//     PlcTask Outputs/GVL_iXlinker.EtherCAT_Master_EPPxxxx.Beckhoff_EPP2xxx.Beckhoff_EPP2xxxEK1122.A_0050_EPP2338_0002_0018.Channel_14.Output <-> Channel 14/Output
//     PlcTask Outputs/GVL_iXlinker.EtherCAT_Master_EPPxxxx.Beckhoff_EPP2xxx.Beckhoff_EPP2xxxEK1122.A_0050_EPP2338_0002_0018.Channel_15.Output <-> Channel 15/Output
//     PlcTask Outputs/GVL_iXlinker.EtherCAT_Master_EPPxxxx.Beckhoff_EPP2xxx.Beckhoff_EPP2xxxEK1122.A_0050_EPP2338_0002_0018.Channel_16.Output <-> Channel 16/Output
//     PlcTask Inputs/GVL_iXlinker.EtherCAT_Master_EPPxxxx.Beckhoff_EPP2xxx.Beckhoff_EPP2xxxEK1122.A_0050_EPP2338_0002_0018.WcState.WcState <-> WcState/WcState
//     PlcTask Inputs/GVL_iXlinker.EtherCAT_Master_EPPxxxx.Beckhoff_EPP2xxx.Beckhoff_EPP2xxxEK1122.A_0050_EPP2338_0002_0018.WcState.InputToggle <-> WcState/InputToggle
//     PlcTask Inputs/GVL_iXlinker.EtherCAT_Master_EPPxxxx.Beckhoff_EPP2xxx.Beckhoff_EPP2xxxEK1122.A_0050_EPP2338_0002_0018.InfoData.State <-> InfoData/State
//   PLC/PLC Instance <-> EtherCAT Master EPPxxxx/Beckhoff EPP2xxx/Beckhoff EPP2xxxEK1122/A_0051(EPP2338-1001-0017)
//     PlcTask Inputs/GVL_iXlinker.EtherCAT_Master_EPPxxxx.Beckhoff_EPP2xxx.Beckhoff_EPP2xxxEK1122.A_0051_EPP2338_1001_0017.Channel_1.Input <-> Channel 1/Input
//     PlcTask Inputs/GVL_iXlinker.EtherCAT_Master_EPPxxxx.Beckhoff_EPP2xxx.Beckhoff_EPP2xxxEK1122.A_0051_EPP2338_1001_0017.Channel_2.Input <-> Channel 2/Input
//     PlcTask Inputs/GVL_iXlinker.EtherCAT_Master_EPPxxxx.Beckhoff_EPP2xxx.Beckhoff_EPP2xxxEK1122.A_0051_EPP2338_1001_0017.Channel_3.Input <-> Channel 3/Input
//     PlcTask Inputs/GVL_iXlinker.EtherCAT_Master_EPPxxxx.Beckhoff_EPP2xxx.Beckhoff_EPP2xxxEK1122.A_0051_EPP2338_1001_0017.Channel_4.Input <-> Channel 4/Input
//     PlcTask Inputs/GVL_iXlinker.EtherCAT_Master_EPPxxxx.Beckhoff_EPP2xxx.Beckhoff_EPP2xxxEK1122.A_0051_EPP2338_1001_0017.Channel_5.Input <-> Channel 5/Input
//     PlcTask Inputs/GVL_iXlinker.EtherCAT_Master_EPPxxxx.Beckhoff_EPP2xxx.Beckhoff_EPP2xxxEK1122.A_0051_EPP2338_1001_0017.Channel_6.Input <-> Channel 6/Input
//     PlcTask Inputs/GVL_iXlinker.EtherCAT_Master_EPPxxxx.Beckhoff_EPP2xxx.Beckhoff_EPP2xxxEK1122.A_0051_EPP2338_1001_0017.Channel_7.Input <-> Channel 7/Input
//     PlcTask Inputs/GVL_iXlinker.EtherCAT_Master_EPPxxxx.Beckhoff_EPP2xxx.Beckhoff_EPP2xxxEK1122.A_0051_EPP2338_1001_0017.Channel_8.Input <-> Channel 8/Input
//     PlcTask Outputs/GVL_iXlinker.EtherCAT_Master_EPPxxxx.Beckhoff_EPP2xxx.Beckhoff_EPP2xxxEK1122.A_0051_EPP2338_1001_0017.Channel_9.Output <-> Channel 9/Output
//     PlcTask Outputs/GVL_iXlinker.EtherCAT_Master_EPPxxxx.Beckhoff_EPP2xxx.Beckhoff_EPP2xxxEK1122.A_0051_EPP2338_1001_0017.Channel_10.Output <-> Channel 10/Output
//     PlcTask Outputs/GVL_iXlinker.EtherCAT_Master_EPPxxxx.Beckhoff_EPP2xxx.Beckhoff_EPP2xxxEK1122.A_0051_EPP2338_1001_0017.Channel_11.Output <-> Channel 11/Output
//     PlcTask Outputs/GVL_iXlinker.EtherCAT_Master_EPPxxxx.Beckhoff_EPP2xxx.Beckhoff_EPP2xxxEK1122.A_0051_EPP2338_1001_0017.Channel_12.Output <-> Channel 12/Output
//     PlcTask Outputs/GVL_iXlinker.EtherCAT_Master_EPPxxxx.Beckhoff_EPP2xxx.Beckhoff_EPP2xxxEK1122.A_0051_EPP2338_1001_0017.Channel_13.Output <-> Channel 13/Output
//     PlcTask Outputs/GVL_iXlinker.EtherCAT_Master_EPPxxxx.Beckhoff_EPP2xxx.Beckhoff_EPP2xxxEK1122.A_0051_EPP2338_1001_0017.Channel_14.Output <-> Channel 14/Output
//     PlcTask Outputs/GVL_iXlinker.EtherCAT_Master_EPPxxxx.Beckhoff_EPP2xxx.Beckhoff_EPP2xxxEK1122.A_0051_EPP2338_1001_0017.Channel_15.Output <-> Channel 15/Output
//     PlcTask Outputs/GVL_iXlinker.EtherCAT_Master_EPPxxxx.Beckhoff_EPP2xxx.Beckhoff_EPP2xxxEK1122.A_0051_EPP2338_1001_0017.Channel_16.Output <-> Channel 16/Output
//     PlcTask Inputs/GVL_iXlinker.EtherCAT_Master_EPPxxxx.Beckhoff_EPP2xxx.Beckhoff_EPP2xxxEK1122.A_0051_EPP2338_1001_0017.WcState.WcState <-> WcState/WcState
//     PlcTask Inputs/GVL_iXlinker.EtherCAT_Master_EPPxxxx.Beckhoff_EPP2xxx.Beckhoff_EPP2xxxEK1122.A_0051_EPP2338_1001_0017.WcState.InputToggle <-> WcState/InputToggle
//     PlcTask Inputs/GVL_iXlinker.EtherCAT_Master_EPPxxxx.Beckhoff_EPP2xxx.Beckhoff_EPP2xxxEK1122.A_0051_EPP2338_1001_0017.InfoData.State <-> InfoData/State
//   PLC/PLC Instance <-> EtherCAT Master EPPxxxx/Beckhoff EPP2xxx/Beckhoff EPP2xxxEK1122/A_0052(EPP2338-1001-0018)
//     PlcTask Inputs/GVL_iXlinker.EtherCAT_Master_EPPxxxx.Beckhoff_EPP2xxx.Beckhoff_EPP2xxxEK1122.A_0052_EPP2338_1001_0018.Channel_1.Input <-> Channel 1/Input
//     PlcTask Inputs/GVL_iXlinker.EtherCAT_Master_EPPxxxx.Beckhoff_EPP2xxx.Beckhoff_EPP2xxxEK1122.A_0052_EPP2338_1001_0018.Channel_2.Input <-> Channel 2/Input
//     PlcTask Inputs/GVL_iXlinker.EtherCAT_Master_EPPxxxx.Beckhoff_EPP2xxx.Beckhoff_EPP2xxxEK1122.A_0052_EPP2338_1001_0018.Channel_3.Input <-> Channel 3/Input
//     PlcTask Inputs/GVL_iXlinker.EtherCAT_Master_EPPxxxx.Beckhoff_EPP2xxx.Beckhoff_EPP2xxxEK1122.A_0052_EPP2338_1001_0018.Channel_4.Input <-> Channel 4/Input
//     PlcTask Inputs/GVL_iXlinker.EtherCAT_Master_EPPxxxx.Beckhoff_EPP2xxx.Beckhoff_EPP2xxxEK1122.A_0052_EPP2338_1001_0018.Channel_5.Input <-> Channel 5/Input
//     PlcTask Inputs/GVL_iXlinker.EtherCAT_Master_EPPxxxx.Beckhoff_EPP2xxx.Beckhoff_EPP2xxxEK1122.A_0052_EPP2338_1001_0018.Channel_6.Input <-> Channel 6/Input
//     PlcTask Inputs/GVL_iXlinker.EtherCAT_Master_EPPxxxx.Beckhoff_EPP2xxx.Beckhoff_EPP2xxxEK1122.A_0052_EPP2338_1001_0018.Channel_7.Input <-> Channel 7/Input
//     PlcTask Inputs/GVL_iXlinker.EtherCAT_Master_EPPxxxx.Beckhoff_EPP2xxx.Beckhoff_EPP2xxxEK1122.A_0052_EPP2338_1001_0018.Channel_8.Input <-> Channel 8/Input
//     PlcTask Outputs/GVL_iXlinker.EtherCAT_Master_EPPxxxx.Beckhoff_EPP2xxx.Beckhoff_EPP2xxxEK1122.A_0052_EPP2338_1001_0018.Channel_9.Output <-> Channel 9/Output
//     PlcTask Outputs/GVL_iXlinker.EtherCAT_Master_EPPxxxx.Beckhoff_EPP2xxx.Beckhoff_EPP2xxxEK1122.A_0052_EPP2338_1001_0018.Channel_10.Output <-> Channel 10/Output
//     PlcTask Outputs/GVL_iXlinker.EtherCAT_Master_EPPxxxx.Beckhoff_EPP2xxx.Beckhoff_EPP2xxxEK1122.A_0052_EPP2338_1001_0018.Channel_11.Output <-> Channel 11/Output
//     PlcTask Outputs/GVL_iXlinker.EtherCAT_Master_EPPxxxx.Beckhoff_EPP2xxx.Beckhoff_EPP2xxxEK1122.A_0052_EPP2338_1001_0018.Channel_12.Output <-> Channel 12/Output
//     PlcTask Outputs/GVL_iXlinker.EtherCAT_Master_EPPxxxx.Beckhoff_EPP2xxx.Beckhoff_EPP2xxxEK1122.A_0052_EPP2338_1001_0018.Channel_13.Output <-> Channel 13/Output
//     PlcTask Outputs/GVL_iXlinker.EtherCAT_Master_EPPxxxx.Beckhoff_EPP2xxx.Beckhoff_EPP2xxxEK1122.A_0052_EPP2338_1001_0018.Channel_14.Output <-> Channel 14/Output
//     PlcTask Outputs/GVL_iXlinker.EtherCAT_Master_EPPxxxx.Beckhoff_EPP2xxx.Beckhoff_EPP2xxxEK1122.A_0052_EPP2338_1001_0018.Channel_15.Output <-> Channel 15/Output
//     PlcTask Outputs/GVL_iXlinker.EtherCAT_Master_EPPxxxx.Beckhoff_EPP2xxx.Beckhoff_EPP2xxxEK1122.A_0052_EPP2338_1001_0018.Channel_16.Output <-> Channel 16/Output
//     PlcTask Inputs/GVL_iXlinker.EtherCAT_Master_EPPxxxx.Beckhoff_EPP2xxx.Beckhoff_EPP2xxxEK1122.A_0052_EPP2338_1001_0018.WcState.WcState <-> WcState/WcState
//     PlcTask Inputs/GVL_iXlinker.EtherCAT_Master_EPPxxxx.Beckhoff_EPP2xxx.Beckhoff_EPP2xxxEK1122.A_0052_EPP2338_1001_0018.WcState.InputToggle <-> WcState/InputToggle
//     PlcTask Inputs/GVL_iXlinker.EtherCAT_Master_EPPxxxx.Beckhoff_EPP2xxx.Beckhoff_EPP2xxxEK1122.A_0052_EPP2338_1001_0018.InfoData.State <-> InfoData/State
//   PLC/PLC Instance <-> EtherCAT Master EPPxxxx/Beckhoff EPP2xxx/Beckhoff EPP2xxxEK1122/A_0053(EPP2338-1001-0019)
//     PlcTask Inputs/GVL_iXlinker.EtherCAT_Master_EPPxxxx.Beckhoff_EPP2xxx.Beckhoff_EPP2xxxEK1122.A_0053_EPP2338_1001_0019.Channel_1.Input <-> Channel 1/Input
//     PlcTask Inputs/GVL_iXlinker.EtherCAT_Master_EPPxxxx.Beckhoff_EPP2xxx.Beckhoff_EPP2xxxEK1122.A_0053_EPP2338_1001_0019.Channel_2.Input <-> Channel 2/Input
//     PlcTask Inputs/GVL_iXlinker.EtherCAT_Master_EPPxxxx.Beckhoff_EPP2xxx.Beckhoff_EPP2xxxEK1122.A_0053_EPP2338_1001_0019.Channel_3.Input <-> Channel 3/Input
//     PlcTask Inputs/GVL_iXlinker.EtherCAT_Master_EPPxxxx.Beckhoff_EPP2xxx.Beckhoff_EPP2xxxEK1122.A_0053_EPP2338_1001_0019.Channel_4.Input <-> Channel 4/Input
//     PlcTask Inputs/GVL_iXlinker.EtherCAT_Master_EPPxxxx.Beckhoff_EPP2xxx.Beckhoff_EPP2xxxEK1122.A_0053_EPP2338_1001_0019.Channel_5.Input <-> Channel 5/Input
//     PlcTask Inputs/GVL_iXlinker.EtherCAT_Master_EPPxxxx.Beckhoff_EPP2xxx.Beckhoff_EPP2xxxEK1122.A_0053_EPP2338_1001_0019.Channel_6.Input <-> Channel 6/Input
//     PlcTask Inputs/GVL_iXlinker.EtherCAT_Master_EPPxxxx.Beckhoff_EPP2xxx.Beckhoff_EPP2xxxEK1122.A_0053_EPP2338_1001_0019.Channel_7.Input <-> Channel 7/Input
//     PlcTask Inputs/GVL_iXlinker.EtherCAT_Master_EPPxxxx.Beckhoff_EPP2xxx.Beckhoff_EPP2xxxEK1122.A_0053_EPP2338_1001_0019.Channel_8.Input <-> Channel 8/Input
//     PlcTask Outputs/GVL_iXlinker.EtherCAT_Master_EPPxxxx.Beckhoff_EPP2xxx.Beckhoff_EPP2xxxEK1122.A_0053_EPP2338_1001_0019.Channel_9.Output <-> Channel 9/Output
//     PlcTask Outputs/GVL_iXlinker.EtherCAT_Master_EPPxxxx.Beckhoff_EPP2xxx.Beckhoff_EPP2xxxEK1122.A_0053_EPP2338_1001_0019.Channel_10.Output <-> Channel 10/Output
//     PlcTask Outputs/GVL_iXlinker.EtherCAT_Master_EPPxxxx.Beckhoff_EPP2xxx.Beckhoff_EPP2xxxEK1122.A_0053_EPP2338_1001_0019.Channel_11.Output <-> Channel 11/Output
//     PlcTask Outputs/GVL_iXlinker.EtherCAT_Master_EPPxxxx.Beckhoff_EPP2xxx.Beckhoff_EPP2xxxEK1122.A_0053_EPP2338_1001_0019.Channel_12.Output <-> Channel 12/Output
//     PlcTask Outputs/GVL_iXlinker.EtherCAT_Master_EPPxxxx.Beckhoff_EPP2xxx.Beckhoff_EPP2xxxEK1122.A_0053_EPP2338_1001_0019.Channel_13.Output <-> Channel 13/Output
//     PlcTask Outputs/GVL_iXlinker.EtherCAT_Master_EPPxxxx.Beckhoff_EPP2xxx.Beckhoff_EPP2xxxEK1122.A_0053_EPP2338_1001_0019.Channel_14.Output <-> Channel 14/Output
//     PlcTask Outputs/GVL_iXlinker.EtherCAT_Master_EPPxxxx.Beckhoff_EPP2xxx.Beckhoff_EPP2xxxEK1122.A_0053_EPP2338_1001_0019.Channel_15.Output <-> Channel 15/Output
//     PlcTask Outputs/GVL_iXlinker.EtherCAT_Master_EPPxxxx.Beckhoff_EPP2xxx.Beckhoff_EPP2xxxEK1122.A_0053_EPP2338_1001_0019.Channel_16.Output <-> Channel 16/Output
//     PlcTask Inputs/GVL_iXlinker.EtherCAT_Master_EPPxxxx.Beckhoff_EPP2xxx.Beckhoff_EPP2xxxEK1122.A_0053_EPP2338_1001_0019.WcState.WcState <-> WcState/WcState
//     PlcTask Inputs/GVL_iXlinker.EtherCAT_Master_EPPxxxx.Beckhoff_EPP2xxx.Beckhoff_EPP2xxxEK1122.A_0053_EPP2338_1001_0019.WcState.InputToggle <-> WcState/InputToggle
//     PlcTask Inputs/GVL_iXlinker.EtherCAT_Master_EPPxxxx.Beckhoff_EPP2xxx.Beckhoff_EPP2xxxEK1122.A_0053_EPP2338_1001_0019.InfoData.State <-> InfoData/State
//   PLC/PLC Instance <-> EtherCAT Master EPPxxxx/Beckhoff EPP2xxx/Beckhoff EPP2xxxEK1122/A_0054(EPP2338-1002-0017)
//     PlcTask Inputs/GVL_iXlinker.EtherCAT_Master_EPPxxxx.Beckhoff_EPP2xxx.Beckhoff_EPP2xxxEK1122.A_0054_EPP2338_1002_0017.Channel_1.Input <-> Channel 1/Input
//     PlcTask Inputs/GVL_iXlinker.EtherCAT_Master_EPPxxxx.Beckhoff_EPP2xxx.Beckhoff_EPP2xxxEK1122.A_0054_EPP2338_1002_0017.Channel_2.Input <-> Channel 2/Input
//     PlcTask Inputs/GVL_iXlinker.EtherCAT_Master_EPPxxxx.Beckhoff_EPP2xxx.Beckhoff_EPP2xxxEK1122.A_0054_EPP2338_1002_0017.Channel_3.Input <-> Channel 3/Input
//     PlcTask Inputs/GVL_iXlinker.EtherCAT_Master_EPPxxxx.Beckhoff_EPP2xxx.Beckhoff_EPP2xxxEK1122.A_0054_EPP2338_1002_0017.Channel_4.Input <-> Channel 4/Input
//     PlcTask Inputs/GVL_iXlinker.EtherCAT_Master_EPPxxxx.Beckhoff_EPP2xxx.Beckhoff_EPP2xxxEK1122.A_0054_EPP2338_1002_0017.Channel_5.Input <-> Channel 5/Input
//     PlcTask Inputs/GVL_iXlinker.EtherCAT_Master_EPPxxxx.Beckhoff_EPP2xxx.Beckhoff_EPP2xxxEK1122.A_0054_EPP2338_1002_0017.Channel_6.Input <-> Channel 6/Input
//     PlcTask Inputs/GVL_iXlinker.EtherCAT_Master_EPPxxxx.Beckhoff_EPP2xxx.Beckhoff_EPP2xxxEK1122.A_0054_EPP2338_1002_0017.Channel_7.Input <-> Channel 7/Input
//     PlcTask Inputs/GVL_iXlinker.EtherCAT_Master_EPPxxxx.Beckhoff_EPP2xxx.Beckhoff_EPP2xxxEK1122.A_0054_EPP2338_1002_0017.Channel_8.Input <-> Channel 8/Input
//     PlcTask Outputs/GVL_iXlinker.EtherCAT_Master_EPPxxxx.Beckhoff_EPP2xxx.Beckhoff_EPP2xxxEK1122.A_0054_EPP2338_1002_0017.Channel_9.Output <-> Channel 9/Output
//     PlcTask Outputs/GVL_iXlinker.EtherCAT_Master_EPPxxxx.Beckhoff_EPP2xxx.Beckhoff_EPP2xxxEK1122.A_0054_EPP2338_1002_0017.Channel_10.Output <-> Channel 10/Output
//     PlcTask Outputs/GVL_iXlinker.EtherCAT_Master_EPPxxxx.Beckhoff_EPP2xxx.Beckhoff_EPP2xxxEK1122.A_0054_EPP2338_1002_0017.Channel_11.Output <-> Channel 11/Output
//     PlcTask Outputs/GVL_iXlinker.EtherCAT_Master_EPPxxxx.Beckhoff_EPP2xxx.Beckhoff_EPP2xxxEK1122.A_0054_EPP2338_1002_0017.Channel_12.Output <-> Channel 12/Output
//     PlcTask Outputs/GVL_iXlinker.EtherCAT_Master_EPPxxxx.Beckhoff_EPP2xxx.Beckhoff_EPP2xxxEK1122.A_0054_EPP2338_1002_0017.Channel_13.Output <-> Channel 13/Output
//     PlcTask Outputs/GVL_iXlinker.EtherCAT_Master_EPPxxxx.Beckhoff_EPP2xxx.Beckhoff_EPP2xxxEK1122.A_0054_EPP2338_1002_0017.Channel_14.Output <-> Channel 14/Output
//     PlcTask Outputs/GVL_iXlinker.EtherCAT_Master_EPPxxxx.Beckhoff_EPP2xxx.Beckhoff_EPP2xxxEK1122.A_0054_EPP2338_1002_0017.Channel_15.Output <-> Channel 15/Output
//     PlcTask Outputs/GVL_iXlinker.EtherCAT_Master_EPPxxxx.Beckhoff_EPP2xxx.Beckhoff_EPP2xxxEK1122.A_0054_EPP2338_1002_0017.Channel_16.Output <-> Channel 16/Output
//     PlcTask Inputs/GVL_iXlinker.EtherCAT_Master_EPPxxxx.Beckhoff_EPP2xxx.Beckhoff_EPP2xxxEK1122.A_0054_EPP2338_1002_0017.WcState.WcState <-> WcState/WcState
//     PlcTask Inputs/GVL_iXlinker.EtherCAT_Master_EPPxxxx.Beckhoff_EPP2xxx.Beckhoff_EPP2xxxEK1122.A_0054_EPP2338_1002_0017.WcState.InputToggle <-> WcState/InputToggle
//     PlcTask Inputs/GVL_iXlinker.EtherCAT_Master_EPPxxxx.Beckhoff_EPP2xxx.Beckhoff_EPP2xxxEK1122.A_0054_EPP2338_1002_0017.InfoData.State <-> InfoData/State
//   PLC/PLC Instance <-> EtherCAT Master EPPxxxx/Beckhoff EPP2xxx/Beckhoff EPP2xxxEK1122/A_0055(EPP2338-1002-0018)
//     PlcTask Inputs/GVL_iXlinker.EtherCAT_Master_EPPxxxx.Beckhoff_EPP2xxx.Beckhoff_EPP2xxxEK1122.A_0055_EPP2338_1002_0018.Channel_1.Input <-> Channel 1/Input
//     PlcTask Inputs/GVL_iXlinker.EtherCAT_Master_EPPxxxx.Beckhoff_EPP2xxx.Beckhoff_EPP2xxxEK1122.A_0055_EPP2338_1002_0018.Channel_2.Input <-> Channel 2/Input
//     PlcTask Inputs/GVL_iXlinker.EtherCAT_Master_EPPxxxx.Beckhoff_EPP2xxx.Beckhoff_EPP2xxxEK1122.A_0055_EPP2338_1002_0018.Channel_3.Input <-> Channel 3/Input
//     PlcTask Inputs/GVL_iXlinker.EtherCAT_Master_EPPxxxx.Beckhoff_EPP2xxx.Beckhoff_EPP2xxxEK1122.A_0055_EPP2338_1002_0018.Channel_4.Input <-> Channel 4/Input
//     PlcTask Inputs/GVL_iXlinker.EtherCAT_Master_EPPxxxx.Beckhoff_EPP2xxx.Beckhoff_EPP2xxxEK1122.A_0055_EPP2338_1002_0018.Channel_5.Input <-> Channel 5/Input
//     PlcTask Inputs/GVL_iXlinker.EtherCAT_Master_EPPxxxx.Beckhoff_EPP2xxx.Beckhoff_EPP2xxxEK1122.A_0055_EPP2338_1002_0018.Channel_6.Input <-> Channel 6/Input
//     PlcTask Inputs/GVL_iXlinker.EtherCAT_Master_EPPxxxx.Beckhoff_EPP2xxx.Beckhoff_EPP2xxxEK1122.A_0055_EPP2338_1002_0018.Channel_7.Input <-> Channel 7/Input
//     PlcTask Inputs/GVL_iXlinker.EtherCAT_Master_EPPxxxx.Beckhoff_EPP2xxx.Beckhoff_EPP2xxxEK1122.A_0055_EPP2338_1002_0018.Channel_8.Input <-> Channel 8/Input
//     PlcTask Outputs/GVL_iXlinker.EtherCAT_Master_EPPxxxx.Beckhoff_EPP2xxx.Beckhoff_EPP2xxxEK1122.A_0055_EPP2338_1002_0018.Channel_9.Output <-> Channel 9/Output
//     PlcTask Outputs/GVL_iXlinker.EtherCAT_Master_EPPxxxx.Beckhoff_EPP2xxx.Beckhoff_EPP2xxxEK1122.A_0055_EPP2338_1002_0018.Channel_10.Output <-> Channel 10/Output
//     PlcTask Outputs/GVL_iXlinker.EtherCAT_Master_EPPxxxx.Beckhoff_EPP2xxx.Beckhoff_EPP2xxxEK1122.A_0055_EPP2338_1002_0018.Channel_11.Output <-> Channel 11/Output
//     PlcTask Outputs/GVL_iXlinker.EtherCAT_Master_EPPxxxx.Beckhoff_EPP2xxx.Beckhoff_EPP2xxxEK1122.A_0055_EPP2338_1002_0018.Channel_12.Output <-> Channel 12/Output
//     PlcTask Outputs/GVL_iXlinker.EtherCAT_Master_EPPxxxx.Beckhoff_EPP2xxx.Beckhoff_EPP2xxxEK1122.A_0055_EPP2338_1002_0018.Channel_13.Output <-> Channel 13/Output
//     PlcTask Outputs/GVL_iXlinker.EtherCAT_Master_EPPxxxx.Beckhoff_EPP2xxx.Beckhoff_EPP2xxxEK1122.A_0055_EPP2338_1002_0018.Channel_14.Output <-> Channel 14/Output
//     PlcTask Outputs/GVL_iXlinker.EtherCAT_Master_EPPxxxx.Beckhoff_EPP2xxx.Beckhoff_EPP2xxxEK1122.A_0055_EPP2338_1002_0018.Channel_15.Output <-> Channel 15/Output
//     PlcTask Outputs/GVL_iXlinker.EtherCAT_Master_EPPxxxx.Beckhoff_EPP2xxx.Beckhoff_EPP2xxxEK1122.A_0055_EPP2338_1002_0018.Channel_16.Output <-> Channel 16/Output
//     PlcTask Inputs/GVL_iXlinker.EtherCAT_Master_EPPxxxx.Beckhoff_EPP2xxx.Beckhoff_EPP2xxxEK1122.A_0055_EPP2338_1002_0018.WcState.WcState <-> WcState/WcState
//     PlcTask Inputs/GVL_iXlinker.EtherCAT_Master_EPPxxxx.Beckhoff_EPP2xxx.Beckhoff_EPP2xxxEK1122.A_0055_EPP2338_1002_0018.WcState.InputToggle <-> WcState/InputToggle
//     PlcTask Inputs/GVL_iXlinker.EtherCAT_Master_EPPxxxx.Beckhoff_EPP2xxx.Beckhoff_EPP2xxxEK1122.A_0055_EPP2338_1002_0018.InfoData.State <-> InfoData/State
//   PLC/PLC Instance <-> EtherCAT Master EPPxxxx/Beckhoff EPP2xxx/Beckhoff EPP2xxxEK1122/A_0056(EPP2338-1002-0019)
//     PlcTask Inputs/GVL_iXlinker.EtherCAT_Master_EPPxxxx.Beckhoff_EPP2xxx.Beckhoff_EPP2xxxEK1122.A_0056_EPP2338_1002_0019.Channel_1.Input <-> Channel 1/Input
//     PlcTask Inputs/GVL_iXlinker.EtherCAT_Master_EPPxxxx.Beckhoff_EPP2xxx.Beckhoff_EPP2xxxEK1122.A_0056_EPP2338_1002_0019.Channel_2.Input <-> Channel 2/Input
//     PlcTask Inputs/GVL_iXlinker.EtherCAT_Master_EPPxxxx.Beckhoff_EPP2xxx.Beckhoff_EPP2xxxEK1122.A_0056_EPP2338_1002_0019.Channel_3.Input <-> Channel 3/Input
//     PlcTask Inputs/GVL_iXlinker.EtherCAT_Master_EPPxxxx.Beckhoff_EPP2xxx.Beckhoff_EPP2xxxEK1122.A_0056_EPP2338_1002_0019.Channel_4.Input <-> Channel 4/Input
//     PlcTask Inputs/GVL_iXlinker.EtherCAT_Master_EPPxxxx.Beckhoff_EPP2xxx.Beckhoff_EPP2xxxEK1122.A_0056_EPP2338_1002_0019.Channel_5.Input <-> Channel 5/Input
//     PlcTask Inputs/GVL_iXlinker.EtherCAT_Master_EPPxxxx.Beckhoff_EPP2xxx.Beckhoff_EPP2xxxEK1122.A_0056_EPP2338_1002_0019.Channel_6.Input <-> Channel 6/Input
//     PlcTask Inputs/GVL_iXlinker.EtherCAT_Master_EPPxxxx.Beckhoff_EPP2xxx.Beckhoff_EPP2xxxEK1122.A_0056_EPP2338_1002_0019.Channel_7.Input <-> Channel 7/Input
//     PlcTask Inputs/GVL_iXlinker.EtherCAT_Master_EPPxxxx.Beckhoff_EPP2xxx.Beckhoff_EPP2xxxEK1122.A_0056_EPP2338_1002_0019.Channel_8.Input <-> Channel 8/Input
//     PlcTask Outputs/GVL_iXlinker.EtherCAT_Master_EPPxxxx.Beckhoff_EPP2xxx.Beckhoff_EPP2xxxEK1122.A_0056_EPP2338_1002_0019.Channel_9.Output <-> Channel 9/Output
//     PlcTask Outputs/GVL_iXlinker.EtherCAT_Master_EPPxxxx.Beckhoff_EPP2xxx.Beckhoff_EPP2xxxEK1122.A_0056_EPP2338_1002_0019.Channel_10.Output <-> Channel 10/Output
//     PlcTask Outputs/GVL_iXlinker.EtherCAT_Master_EPPxxxx.Beckhoff_EPP2xxx.Beckhoff_EPP2xxxEK1122.A_0056_EPP2338_1002_0019.Channel_11.Output <-> Channel 11/Output
//     PlcTask Outputs/GVL_iXlinker.EtherCAT_Master_EPPxxxx.Beckhoff_EPP2xxx.Beckhoff_EPP2xxxEK1122.A_0056_EPP2338_1002_0019.Channel_12.Output <-> Channel 12/Output
//     PlcTask Outputs/GVL_iXlinker.EtherCAT_Master_EPPxxxx.Beckhoff_EPP2xxx.Beckhoff_EPP2xxxEK1122.A_0056_EPP2338_1002_0019.Channel_13.Output <-> Channel 13/Output
//     PlcTask Outputs/GVL_iXlinker.EtherCAT_Master_EPPxxxx.Beckhoff_EPP2xxx.Beckhoff_EPP2xxxEK1122.A_0056_EPP2338_1002_0019.Channel_14.Output <-> Channel 14/Output
//     PlcTask Outputs/GVL_iXlinker.EtherCAT_Master_EPPxxxx.Beckhoff_EPP2xxx.Beckhoff_EPP2xxxEK1122.A_0056_EPP2338_1002_0019.Channel_15.Output <-> Channel 15/Output
//     PlcTask Outputs/GVL_iXlinker.EtherCAT_Master_EPPxxxx.Beckhoff_EPP2xxx.Beckhoff_EPP2xxxEK1122.A_0056_EPP2338_1002_0019.Channel_16.Output <-> Channel 16/Output
//     PlcTask Inputs/GVL_iXlinker.EtherCAT_Master_EPPxxxx.Beckhoff_EPP2xxx.Beckhoff_EPP2xxxEK1122.A_0056_EPP2338_1002_0019.WcState.WcState <-> WcState/WcState
//     PlcTask Inputs/GVL_iXlinker.EtherCAT_Master_EPPxxxx.Beckhoff_EPP2xxx.Beckhoff_EPP2xxxEK1122.A_0056_EPP2338_1002_0019.WcState.InputToggle <-> WcState/InputToggle
//     PlcTask Inputs/GVL_iXlinker.EtherCAT_Master_EPPxxxx.Beckhoff_EPP2xxx.Beckhoff_EPP2xxxEK1122.A_0056_EPP2338_1002_0019.InfoData.State <-> InfoData/State
//   PLC/PLC Instance <-> EtherCAT Master EPPxxxx/Beckhoff EPP2xxx/Beckhoff EPP2xxxEK1122/A_0057(EPP2339-0003-0016)
//     PlcTask Inputs/GVL_iXlinker.EtherCAT_Master_EPPxxxx.Beckhoff_EPP2xxx.Beckhoff_EPP2xxxEK1122.A_0057_EPP2339_0003_0016.DI_Inputs_Channel_1.Input[0] <-> DI Inputs Channel 1/Input 1
//     PlcTask Inputs/GVL_iXlinker.EtherCAT_Master_EPPxxxx.Beckhoff_EPP2xxx.Beckhoff_EPP2xxxEK1122.A_0057_EPP2339_0003_0016.DI_Inputs_Channel_1.Input[1] <-> DI Inputs Channel 1/Input 2
//     PlcTask Inputs/GVL_iXlinker.EtherCAT_Master_EPPxxxx.Beckhoff_EPP2xxx.Beckhoff_EPP2xxxEK1122.A_0057_EPP2339_0003_0016.DI_Inputs_Channel_1.Input[2] <-> DI Inputs Channel 1/Input 3
//     PlcTask Inputs/GVL_iXlinker.EtherCAT_Master_EPPxxxx.Beckhoff_EPP2xxx.Beckhoff_EPP2xxxEK1122.A_0057_EPP2339_0003_0016.DI_Inputs_Channel_1.Input[3] <-> DI Inputs Channel 1/Input 4
//     PlcTask Inputs/GVL_iXlinker.EtherCAT_Master_EPPxxxx.Beckhoff_EPP2xxx.Beckhoff_EPP2xxxEK1122.A_0057_EPP2339_0003_0016.DI_Inputs_Channel_1.Input[4] <-> DI Inputs Channel 1/Input 5
//     PlcTask Inputs/GVL_iXlinker.EtherCAT_Master_EPPxxxx.Beckhoff_EPP2xxx.Beckhoff_EPP2xxxEK1122.A_0057_EPP2339_0003_0016.DI_Inputs_Channel_1.Input[5] <-> DI Inputs Channel 1/Input 6
//     PlcTask Inputs/GVL_iXlinker.EtherCAT_Master_EPPxxxx.Beckhoff_EPP2xxx.Beckhoff_EPP2xxxEK1122.A_0057_EPP2339_0003_0016.DI_Inputs_Channel_1.Input[6] <-> DI Inputs Channel 1/Input 7
//     PlcTask Inputs/GVL_iXlinker.EtherCAT_Master_EPPxxxx.Beckhoff_EPP2xxx.Beckhoff_EPP2xxxEK1122.A_0057_EPP2339_0003_0016.DI_Inputs_Channel_1.Input[7] <-> DI Inputs Channel 1/Input 8
//     PlcTask Inputs/GVL_iXlinker.EtherCAT_Master_EPPxxxx.Beckhoff_EPP2xxx.Beckhoff_EPP2xxxEK1122.A_0057_EPP2339_0003_0016.DI_Inputs_Channel_2.Input[0] <-> DI Inputs Channel 2/Input 1
//     PlcTask Inputs/GVL_iXlinker.EtherCAT_Master_EPPxxxx.Beckhoff_EPP2xxx.Beckhoff_EPP2xxxEK1122.A_0057_EPP2339_0003_0016.DI_Inputs_Channel_2.Input[1] <-> DI Inputs Channel 2/Input 2
//     PlcTask Inputs/GVL_iXlinker.EtherCAT_Master_EPPxxxx.Beckhoff_EPP2xxx.Beckhoff_EPP2xxxEK1122.A_0057_EPP2339_0003_0016.DI_Inputs_Channel_2.Input[2] <-> DI Inputs Channel 2/Input 3
//     PlcTask Inputs/GVL_iXlinker.EtherCAT_Master_EPPxxxx.Beckhoff_EPP2xxx.Beckhoff_EPP2xxxEK1122.A_0057_EPP2339_0003_0016.DI_Inputs_Channel_2.Input[3] <-> DI Inputs Channel 2/Input 4
//     PlcTask Inputs/GVL_iXlinker.EtherCAT_Master_EPPxxxx.Beckhoff_EPP2xxx.Beckhoff_EPP2xxxEK1122.A_0057_EPP2339_0003_0016.DI_Inputs_Channel_2.Input[4] <-> DI Inputs Channel 2/Input 5
//     PlcTask Inputs/GVL_iXlinker.EtherCAT_Master_EPPxxxx.Beckhoff_EPP2xxx.Beckhoff_EPP2xxxEK1122.A_0057_EPP2339_0003_0016.DI_Inputs_Channel_2.Input[5] <-> DI Inputs Channel 2/Input 6
//     PlcTask Inputs/GVL_iXlinker.EtherCAT_Master_EPPxxxx.Beckhoff_EPP2xxx.Beckhoff_EPP2xxxEK1122.A_0057_EPP2339_0003_0016.DI_Inputs_Channel_2.Input[6] <-> DI Inputs Channel 2/Input 7
//     PlcTask Inputs/GVL_iXlinker.EtherCAT_Master_EPPxxxx.Beckhoff_EPP2xxx.Beckhoff_EPP2xxxEK1122.A_0057_EPP2339_0003_0016.DI_Inputs_Channel_2.Input[7] <-> DI Inputs Channel 2/Input 8
//     PlcTask Inputs/GVL_iXlinker.EtherCAT_Master_EPPxxxx.Beckhoff_EPP2xxx.Beckhoff_EPP2xxxEK1122.A_0057_EPP2339_0003_0016.DI_Inputs_Channel_1.Sync_error <-> DI Inputs Channel 1/Sync error
//     PlcTask Inputs/GVL_iXlinker.EtherCAT_Master_EPPxxxx.Beckhoff_EPP2xxx.Beckhoff_EPP2xxxEK1122.A_0057_EPP2339_0003_0016.DI_Inputs_Channel_2.Sync_error <-> DI Inputs Channel 2/Sync error
//     PlcTask Inputs/GVL_iXlinker.EtherCAT_Master_EPPxxxx.Beckhoff_EPP2xxx.Beckhoff_EPP2xxxEK1122.A_0057_EPP2339_0003_0016.DI_Inputs_Channel_1.TxPDO_State <-> DI Inputs Channel 1/TxPDO State
//     PlcTask Inputs/GVL_iXlinker.EtherCAT_Master_EPPxxxx.Beckhoff_EPP2xxx.Beckhoff_EPP2xxxEK1122.A_0057_EPP2339_0003_0016.DI_Inputs_Channel_2.TxPDO_State <-> DI Inputs Channel 2/TxPDO State
//     PlcTask Inputs/GVL_iXlinker.EtherCAT_Master_EPPxxxx.Beckhoff_EPP2xxx.Beckhoff_EPP2xxxEK1122.A_0057_EPP2339_0003_0016.DI_Inputs_Channel_1.TxPDO_Toggle <-> DI Inputs Channel 1/TxPDO Toggle
//     PlcTask Inputs/GVL_iXlinker.EtherCAT_Master_EPPxxxx.Beckhoff_EPP2xxx.Beckhoff_EPP2xxxEK1122.A_0057_EPP2339_0003_0016.DI_Inputs_Channel_2.TxPDO_Toggle <-> DI Inputs Channel 2/TxPDO Toggle
//     PlcTask Outputs/GVL_iXlinker.EtherCAT_Master_EPPxxxx.Beckhoff_EPP2xxx.Beckhoff_EPP2xxxEK1122.A_0057_EPP2339_0003_0016.DO_Outputs_Channel_1.Output[0] <-> DO Outputs Channel 1/Output 1
//     PlcTask Outputs/GVL_iXlinker.EtherCAT_Master_EPPxxxx.Beckhoff_EPP2xxx.Beckhoff_EPP2xxxEK1122.A_0057_EPP2339_0003_0016.DO_Outputs_Channel_1.Output[1] <-> DO Outputs Channel 1/Output 2
//     PlcTask Outputs/GVL_iXlinker.EtherCAT_Master_EPPxxxx.Beckhoff_EPP2xxx.Beckhoff_EPP2xxxEK1122.A_0057_EPP2339_0003_0016.DO_Outputs_Channel_1.Output[2] <-> DO Outputs Channel 1/Output 3
//     PlcTask Outputs/GVL_iXlinker.EtherCAT_Master_EPPxxxx.Beckhoff_EPP2xxx.Beckhoff_EPP2xxxEK1122.A_0057_EPP2339_0003_0016.DO_Outputs_Channel_1.Output[3] <-> DO Outputs Channel 1/Output 4
//     PlcTask Outputs/GVL_iXlinker.EtherCAT_Master_EPPxxxx.Beckhoff_EPP2xxx.Beckhoff_EPP2xxxEK1122.A_0057_EPP2339_0003_0016.DO_Outputs_Channel_1.Output[4] <-> DO Outputs Channel 1/Output 5
//     PlcTask Outputs/GVL_iXlinker.EtherCAT_Master_EPPxxxx.Beckhoff_EPP2xxx.Beckhoff_EPP2xxxEK1122.A_0057_EPP2339_0003_0016.DO_Outputs_Channel_1.Output[5] <-> DO Outputs Channel 1/Output 6
//     PlcTask Outputs/GVL_iXlinker.EtherCAT_Master_EPPxxxx.Beckhoff_EPP2xxx.Beckhoff_EPP2xxxEK1122.A_0057_EPP2339_0003_0016.DO_Outputs_Channel_1.Output[6] <-> DO Outputs Channel 1/Output 7
//     PlcTask Outputs/GVL_iXlinker.EtherCAT_Master_EPPxxxx.Beckhoff_EPP2xxx.Beckhoff_EPP2xxxEK1122.A_0057_EPP2339_0003_0016.DO_Outputs_Channel_1.Output[7] <-> DO Outputs Channel 1/Output 8
//     PlcTask Outputs/GVL_iXlinker.EtherCAT_Master_EPPxxxx.Beckhoff_EPP2xxx.Beckhoff_EPP2xxxEK1122.A_0057_EPP2339_0003_0016.DO_Outputs_Channel_2.Output[0] <-> DO Outputs Channel 2/Output 1
//     PlcTask Outputs/GVL_iXlinker.EtherCAT_Master_EPPxxxx.Beckhoff_EPP2xxx.Beckhoff_EPP2xxxEK1122.A_0057_EPP2339_0003_0016.DO_Outputs_Channel_2.Output[1] <-> DO Outputs Channel 2/Output 2
//     PlcTask Outputs/GVL_iXlinker.EtherCAT_Master_EPPxxxx.Beckhoff_EPP2xxx.Beckhoff_EPP2xxxEK1122.A_0057_EPP2339_0003_0016.DO_Outputs_Channel_2.Output[2] <-> DO Outputs Channel 2/Output 3
//     PlcTask Outputs/GVL_iXlinker.EtherCAT_Master_EPPxxxx.Beckhoff_EPP2xxx.Beckhoff_EPP2xxxEK1122.A_0057_EPP2339_0003_0016.DO_Outputs_Channel_2.Output[3] <-> DO Outputs Channel 2/Output 4
//     PlcTask Outputs/GVL_iXlinker.EtherCAT_Master_EPPxxxx.Beckhoff_EPP2xxx.Beckhoff_EPP2xxxEK1122.A_0057_EPP2339_0003_0016.DO_Outputs_Channel_2.Output[4] <-> DO Outputs Channel 2/Output 5
//     PlcTask Outputs/GVL_iXlinker.EtherCAT_Master_EPPxxxx.Beckhoff_EPP2xxx.Beckhoff_EPP2xxxEK1122.A_0057_EPP2339_0003_0016.DO_Outputs_Channel_2.Output[5] <-> DO Outputs Channel 2/Output 6
//     PlcTask Outputs/GVL_iXlinker.EtherCAT_Master_EPPxxxx.Beckhoff_EPP2xxx.Beckhoff_EPP2xxxEK1122.A_0057_EPP2339_0003_0016.DO_Outputs_Channel_2.Output[6] <-> DO Outputs Channel 2/Output 7
//     PlcTask Outputs/GVL_iXlinker.EtherCAT_Master_EPPxxxx.Beckhoff_EPP2xxx.Beckhoff_EPP2xxxEK1122.A_0057_EPP2339_0003_0016.DO_Outputs_Channel_2.Output[7] <-> DO Outputs Channel 2/Output 8
//     PlcTask Inputs/GVL_iXlinker.EtherCAT_Master_EPPxxxx.Beckhoff_EPP2xxx.Beckhoff_EPP2xxxEK1122.A_0057_EPP2339_0003_0016.WcState.WcState <-> WcState/WcState
//     PlcTask Inputs/GVL_iXlinker.EtherCAT_Master_EPPxxxx.Beckhoff_EPP2xxx.Beckhoff_EPP2xxxEK1122.A_0057_EPP2339_0003_0016.WcState.InputToggle <-> WcState/InputToggle
//     PlcTask Inputs/GVL_iXlinker.EtherCAT_Master_EPPxxxx.Beckhoff_EPP2xxx.Beckhoff_EPP2xxxEK1122.A_0057_EPP2339_0003_0016.InfoData.AdsAddr <-> InfoData/AdsAddr
//     PlcTask Inputs/GVL_iXlinker.EtherCAT_Master_EPPxxxx.Beckhoff_EPP2xxx.Beckhoff_EPP2xxxEK1122.A_0057_EPP2339_0003_0016.InfoData.State <-> InfoData/State
//   PLC/PLC Instance <-> EtherCAT Master EPPxxxx/Beckhoff EPP2xxx/Beckhoff EPP2xxxEK1122/A_0058(EPP2339-0021-0016)
//     PlcTask Inputs/GVL_iXlinker.EtherCAT_Master_EPPxxxx.Beckhoff_EPP2xxx.Beckhoff_EPP2xxxEK1122.A_0058_EPP2339_0021_0016.Channel_1.Input <-> Channel 1/Input
//     PlcTask Inputs/GVL_iXlinker.EtherCAT_Master_EPPxxxx.Beckhoff_EPP2xxx.Beckhoff_EPP2xxxEK1122.A_0058_EPP2339_0021_0016.Channel_2.Input <-> Channel 2/Input
//     PlcTask Inputs/GVL_iXlinker.EtherCAT_Master_EPPxxxx.Beckhoff_EPP2xxx.Beckhoff_EPP2xxxEK1122.A_0058_EPP2339_0021_0016.Channel_3.Input <-> Channel 3/Input
//     PlcTask Inputs/GVL_iXlinker.EtherCAT_Master_EPPxxxx.Beckhoff_EPP2xxx.Beckhoff_EPP2xxxEK1122.A_0058_EPP2339_0021_0016.Channel_4.Input <-> Channel 4/Input
//     PlcTask Inputs/GVL_iXlinker.EtherCAT_Master_EPPxxxx.Beckhoff_EPP2xxx.Beckhoff_EPP2xxxEK1122.A_0058_EPP2339_0021_0016.Channel_5.Input <-> Channel 5/Input
//     PlcTask Inputs/GVL_iXlinker.EtherCAT_Master_EPPxxxx.Beckhoff_EPP2xxx.Beckhoff_EPP2xxxEK1122.A_0058_EPP2339_0021_0016.Channel_6.Input <-> Channel 6/Input
//     PlcTask Inputs/GVL_iXlinker.EtherCAT_Master_EPPxxxx.Beckhoff_EPP2xxx.Beckhoff_EPP2xxxEK1122.A_0058_EPP2339_0021_0016.Channel_7.Input <-> Channel 7/Input
//     PlcTask Inputs/GVL_iXlinker.EtherCAT_Master_EPPxxxx.Beckhoff_EPP2xxx.Beckhoff_EPP2xxxEK1122.A_0058_EPP2339_0021_0016.Channel_8.Input <-> Channel 8/Input
//     PlcTask Inputs/GVL_iXlinker.EtherCAT_Master_EPPxxxx.Beckhoff_EPP2xxx.Beckhoff_EPP2xxxEK1122.A_0058_EPP2339_0021_0016.Channel_9.Input <-> Channel 9/Input
//     PlcTask Inputs/GVL_iXlinker.EtherCAT_Master_EPPxxxx.Beckhoff_EPP2xxx.Beckhoff_EPP2xxxEK1122.A_0058_EPP2339_0021_0016.Channel_10.Input <-> Channel 10/Input
//     PlcTask Inputs/GVL_iXlinker.EtherCAT_Master_EPPxxxx.Beckhoff_EPP2xxx.Beckhoff_EPP2xxxEK1122.A_0058_EPP2339_0021_0016.Channel_11.Input <-> Channel 11/Input
//     PlcTask Inputs/GVL_iXlinker.EtherCAT_Master_EPPxxxx.Beckhoff_EPP2xxx.Beckhoff_EPP2xxxEK1122.A_0058_EPP2339_0021_0016.Channel_12.Input <-> Channel 12/Input
//     PlcTask Inputs/GVL_iXlinker.EtherCAT_Master_EPPxxxx.Beckhoff_EPP2xxx.Beckhoff_EPP2xxxEK1122.A_0058_EPP2339_0021_0016.Channel_13.Input <-> Channel 13/Input
//     PlcTask Inputs/GVL_iXlinker.EtherCAT_Master_EPPxxxx.Beckhoff_EPP2xxx.Beckhoff_EPP2xxxEK1122.A_0058_EPP2339_0021_0016.Channel_14.Input <-> Channel 14/Input
//     PlcTask Inputs/GVL_iXlinker.EtherCAT_Master_EPPxxxx.Beckhoff_EPP2xxx.Beckhoff_EPP2xxxEK1122.A_0058_EPP2339_0021_0016.Channel_15.Input <-> Channel 15/Input
//     PlcTask Inputs/GVL_iXlinker.EtherCAT_Master_EPPxxxx.Beckhoff_EPP2xxx.Beckhoff_EPP2xxxEK1122.A_0058_EPP2339_0021_0016.Channel_16.Input <-> Channel 16/Input
//     PlcTask Outputs/GVL_iXlinker.EtherCAT_Master_EPPxxxx.Beckhoff_EPP2xxx.Beckhoff_EPP2xxxEK1122.A_0058_EPP2339_0021_0016.Channel_9_1.Output <-> Channel 9_1/Output
//     PlcTask Outputs/GVL_iXlinker.EtherCAT_Master_EPPxxxx.Beckhoff_EPP2xxx.Beckhoff_EPP2xxxEK1122.A_0058_EPP2339_0021_0016.Channel_10_1.Output <-> Channel 10_1/Output
//     PlcTask Outputs/GVL_iXlinker.EtherCAT_Master_EPPxxxx.Beckhoff_EPP2xxx.Beckhoff_EPP2xxxEK1122.A_0058_EPP2339_0021_0016.Channel_11_1.Output <-> Channel 11_1/Output
//     PlcTask Outputs/GVL_iXlinker.EtherCAT_Master_EPPxxxx.Beckhoff_EPP2xxx.Beckhoff_EPP2xxxEK1122.A_0058_EPP2339_0021_0016.Channel_12_1.Output <-> Channel 12_1/Output
//     PlcTask Outputs/GVL_iXlinker.EtherCAT_Master_EPPxxxx.Beckhoff_EPP2xxx.Beckhoff_EPP2xxxEK1122.A_0058_EPP2339_0021_0016.Channel_13_1.Output <-> Channel 13_1/Output
//     PlcTask Outputs/GVL_iXlinker.EtherCAT_Master_EPPxxxx.Beckhoff_EPP2xxx.Beckhoff_EPP2xxxEK1122.A_0058_EPP2339_0021_0016.Channel_14_1.Output <-> Channel 14_1/Output
//     PlcTask Outputs/GVL_iXlinker.EtherCAT_Master_EPPxxxx.Beckhoff_EPP2xxx.Beckhoff_EPP2xxxEK1122.A_0058_EPP2339_0021_0016.Channel_15_1.Output <-> Channel 15_1/Output
//     PlcTask Outputs/GVL_iXlinker.EtherCAT_Master_EPPxxxx.Beckhoff_EPP2xxx.Beckhoff_EPP2xxxEK1122.A_0058_EPP2339_0021_0016.Channel_16_1.Output <-> Channel 16_1/Output
//     PlcTask Outputs/GVL_iXlinker.EtherCAT_Master_EPPxxxx.Beckhoff_EPP2xxx.Beckhoff_EPP2xxxEK1122.A_0058_EPP2339_0021_0016.Channel_25.Output <-> Channel 25/Output
//     PlcTask Outputs/GVL_iXlinker.EtherCAT_Master_EPPxxxx.Beckhoff_EPP2xxx.Beckhoff_EPP2xxxEK1122.A_0058_EPP2339_0021_0016.Channel_26.Output <-> Channel 26/Output
//     PlcTask Outputs/GVL_iXlinker.EtherCAT_Master_EPPxxxx.Beckhoff_EPP2xxx.Beckhoff_EPP2xxxEK1122.A_0058_EPP2339_0021_0016.Channel_27.Output <-> Channel 27/Output
//     PlcTask Outputs/GVL_iXlinker.EtherCAT_Master_EPPxxxx.Beckhoff_EPP2xxx.Beckhoff_EPP2xxxEK1122.A_0058_EPP2339_0021_0016.Channel_28.Output <-> Channel 28/Output
//     PlcTask Outputs/GVL_iXlinker.EtherCAT_Master_EPPxxxx.Beckhoff_EPP2xxx.Beckhoff_EPP2xxxEK1122.A_0058_EPP2339_0021_0016.Channel_29.Output <-> Channel 29/Output
//     PlcTask Outputs/GVL_iXlinker.EtherCAT_Master_EPPxxxx.Beckhoff_EPP2xxx.Beckhoff_EPP2xxxEK1122.A_0058_EPP2339_0021_0016.Channel_30.Output <-> Channel 30/Output
//     PlcTask Outputs/GVL_iXlinker.EtherCAT_Master_EPPxxxx.Beckhoff_EPP2xxx.Beckhoff_EPP2xxxEK1122.A_0058_EPP2339_0021_0016.Channel_31.Output <-> Channel 31/Output
//     PlcTask Outputs/GVL_iXlinker.EtherCAT_Master_EPPxxxx.Beckhoff_EPP2xxx.Beckhoff_EPP2xxxEK1122.A_0058_EPP2339_0021_0016.Channel_32.Output <-> Channel 32/Output
//     PlcTask Inputs/GVL_iXlinker.EtherCAT_Master_EPPxxxx.Beckhoff_EPP2xxx.Beckhoff_EPP2xxxEK1122.A_0058_EPP2339_0021_0016.WcState.WcState <-> WcState/WcState
//     PlcTask Inputs/GVL_iXlinker.EtherCAT_Master_EPPxxxx.Beckhoff_EPP2xxx.Beckhoff_EPP2xxxEK1122.A_0058_EPP2339_0021_0016.WcState.InputToggle <-> WcState/InputToggle
//     PlcTask Inputs/GVL_iXlinker.EtherCAT_Master_EPPxxxx.Beckhoff_EPP2xxx.Beckhoff_EPP2xxxEK1122.A_0058_EPP2339_0021_0016.InfoData.State <-> InfoData/State
//   PLC/PLC Instance <-> EtherCAT Master EPPxxxx/Beckhoff EPP2xxx/Beckhoff EPP2xxxEK1122/A_0059(EPP2339-0021-0017)
//     PlcTask Inputs/GVL_iXlinker.EtherCAT_Master_EPPxxxx.Beckhoff_EPP2xxx.Beckhoff_EPP2xxxEK1122.A_0059_EPP2339_0021_0017.Channel_1.Input <-> Channel 1/Input
//     PlcTask Inputs/GVL_iXlinker.EtherCAT_Master_EPPxxxx.Beckhoff_EPP2xxx.Beckhoff_EPP2xxxEK1122.A_0059_EPP2339_0021_0017.Channel_2.Input <-> Channel 2/Input
//     PlcTask Inputs/GVL_iXlinker.EtherCAT_Master_EPPxxxx.Beckhoff_EPP2xxx.Beckhoff_EPP2xxxEK1122.A_0059_EPP2339_0021_0017.Channel_3.Input <-> Channel 3/Input
//     PlcTask Inputs/GVL_iXlinker.EtherCAT_Master_EPPxxxx.Beckhoff_EPP2xxx.Beckhoff_EPP2xxxEK1122.A_0059_EPP2339_0021_0017.Channel_4.Input <-> Channel 4/Input
//     PlcTask Inputs/GVL_iXlinker.EtherCAT_Master_EPPxxxx.Beckhoff_EPP2xxx.Beckhoff_EPP2xxxEK1122.A_0059_EPP2339_0021_0017.Channel_5.Input <-> Channel 5/Input
//     PlcTask Inputs/GVL_iXlinker.EtherCAT_Master_EPPxxxx.Beckhoff_EPP2xxx.Beckhoff_EPP2xxxEK1122.A_0059_EPP2339_0021_0017.Channel_6.Input <-> Channel 6/Input
//     PlcTask Inputs/GVL_iXlinker.EtherCAT_Master_EPPxxxx.Beckhoff_EPP2xxx.Beckhoff_EPP2xxxEK1122.A_0059_EPP2339_0021_0017.Channel_7.Input <-> Channel 7/Input
//     PlcTask Inputs/GVL_iXlinker.EtherCAT_Master_EPPxxxx.Beckhoff_EPP2xxx.Beckhoff_EPP2xxxEK1122.A_0059_EPP2339_0021_0017.Channel_8.Input <-> Channel 8/Input
//     PlcTask Inputs/GVL_iXlinker.EtherCAT_Master_EPPxxxx.Beckhoff_EPP2xxx.Beckhoff_EPP2xxxEK1122.A_0059_EPP2339_0021_0017.Channel_9.Input <-> Channel 9/Input
//     PlcTask Inputs/GVL_iXlinker.EtherCAT_Master_EPPxxxx.Beckhoff_EPP2xxx.Beckhoff_EPP2xxxEK1122.A_0059_EPP2339_0021_0017.Channel_10.Input <-> Channel 10/Input
//     PlcTask Inputs/GVL_iXlinker.EtherCAT_Master_EPPxxxx.Beckhoff_EPP2xxx.Beckhoff_EPP2xxxEK1122.A_0059_EPP2339_0021_0017.Channel_11.Input <-> Channel 11/Input
//     PlcTask Inputs/GVL_iXlinker.EtherCAT_Master_EPPxxxx.Beckhoff_EPP2xxx.Beckhoff_EPP2xxxEK1122.A_0059_EPP2339_0021_0017.Channel_12.Input <-> Channel 12/Input
//     PlcTask Inputs/GVL_iXlinker.EtherCAT_Master_EPPxxxx.Beckhoff_EPP2xxx.Beckhoff_EPP2xxxEK1122.A_0059_EPP2339_0021_0017.Channel_13.Input <-> Channel 13/Input
//     PlcTask Inputs/GVL_iXlinker.EtherCAT_Master_EPPxxxx.Beckhoff_EPP2xxx.Beckhoff_EPP2xxxEK1122.A_0059_EPP2339_0021_0017.Channel_14.Input <-> Channel 14/Input
//     PlcTask Inputs/GVL_iXlinker.EtherCAT_Master_EPPxxxx.Beckhoff_EPP2xxx.Beckhoff_EPP2xxxEK1122.A_0059_EPP2339_0021_0017.Channel_15.Input <-> Channel 15/Input
//     PlcTask Inputs/GVL_iXlinker.EtherCAT_Master_EPPxxxx.Beckhoff_EPP2xxx.Beckhoff_EPP2xxxEK1122.A_0059_EPP2339_0021_0017.Channel_16.Input <-> Channel 16/Input
//     PlcTask Outputs/GVL_iXlinker.EtherCAT_Master_EPPxxxx.Beckhoff_EPP2xxx.Beckhoff_EPP2xxxEK1122.A_0059_EPP2339_0021_0017.Channel_17.Output <-> Channel 17/Output
//     PlcTask Outputs/GVL_iXlinker.EtherCAT_Master_EPPxxxx.Beckhoff_EPP2xxx.Beckhoff_EPP2xxxEK1122.A_0059_EPP2339_0021_0017.Channel_18.Output <-> Channel 18/Output
//     PlcTask Outputs/GVL_iXlinker.EtherCAT_Master_EPPxxxx.Beckhoff_EPP2xxx.Beckhoff_EPP2xxxEK1122.A_0059_EPP2339_0021_0017.Channel_19.Output <-> Channel 19/Output
//     PlcTask Outputs/GVL_iXlinker.EtherCAT_Master_EPPxxxx.Beckhoff_EPP2xxx.Beckhoff_EPP2xxxEK1122.A_0059_EPP2339_0021_0017.Channel_20.Output <-> Channel 20/Output
//     PlcTask Outputs/GVL_iXlinker.EtherCAT_Master_EPPxxxx.Beckhoff_EPP2xxx.Beckhoff_EPP2xxxEK1122.A_0059_EPP2339_0021_0017.Channel_21.Output <-> Channel 21/Output
//     PlcTask Outputs/GVL_iXlinker.EtherCAT_Master_EPPxxxx.Beckhoff_EPP2xxx.Beckhoff_EPP2xxxEK1122.A_0059_EPP2339_0021_0017.Channel_22.Output <-> Channel 22/Output
//     PlcTask Outputs/GVL_iXlinker.EtherCAT_Master_EPPxxxx.Beckhoff_EPP2xxx.Beckhoff_EPP2xxxEK1122.A_0059_EPP2339_0021_0017.Channel_23.Output <-> Channel 23/Output
//     PlcTask Outputs/GVL_iXlinker.EtherCAT_Master_EPPxxxx.Beckhoff_EPP2xxx.Beckhoff_EPP2xxxEK1122.A_0059_EPP2339_0021_0017.Channel_24.Output <-> Channel 24/Output
//     PlcTask Outputs/GVL_iXlinker.EtherCAT_Master_EPPxxxx.Beckhoff_EPP2xxx.Beckhoff_EPP2xxxEK1122.A_0059_EPP2339_0021_0017.Channel_25.Output <-> Channel 25/Output
//     PlcTask Outputs/GVL_iXlinker.EtherCAT_Master_EPPxxxx.Beckhoff_EPP2xxx.Beckhoff_EPP2xxxEK1122.A_0059_EPP2339_0021_0017.Channel_26.Output <-> Channel 26/Output
//     PlcTask Outputs/GVL_iXlinker.EtherCAT_Master_EPPxxxx.Beckhoff_EPP2xxx.Beckhoff_EPP2xxxEK1122.A_0059_EPP2339_0021_0017.Channel_27.Output <-> Channel 27/Output
//     PlcTask Outputs/GVL_iXlinker.EtherCAT_Master_EPPxxxx.Beckhoff_EPP2xxx.Beckhoff_EPP2xxxEK1122.A_0059_EPP2339_0021_0017.Channel_28.Output <-> Channel 28/Output
//     PlcTask Outputs/GVL_iXlinker.EtherCAT_Master_EPPxxxx.Beckhoff_EPP2xxx.Beckhoff_EPP2xxxEK1122.A_0059_EPP2339_0021_0017.Channel_29.Output <-> Channel 29/Output
//     PlcTask Outputs/GVL_iXlinker.EtherCAT_Master_EPPxxxx.Beckhoff_EPP2xxx.Beckhoff_EPP2xxxEK1122.A_0059_EPP2339_0021_0017.Channel_30.Output <-> Channel 30/Output
//     PlcTask Outputs/GVL_iXlinker.EtherCAT_Master_EPPxxxx.Beckhoff_EPP2xxx.Beckhoff_EPP2xxxEK1122.A_0059_EPP2339_0021_0017.Channel_31.Output <-> Channel 31/Output
//     PlcTask Outputs/GVL_iXlinker.EtherCAT_Master_EPPxxxx.Beckhoff_EPP2xxx.Beckhoff_EPP2xxxEK1122.A_0059_EPP2339_0021_0017.Channel_32.Output <-> Channel 32/Output
//     PlcTask Inputs/GVL_iXlinker.EtherCAT_Master_EPPxxxx.Beckhoff_EPP2xxx.Beckhoff_EPP2xxxEK1122.A_0059_EPP2339_0021_0017.WcState.WcState <-> WcState/WcState
//     PlcTask Inputs/GVL_iXlinker.EtherCAT_Master_EPPxxxx.Beckhoff_EPP2xxx.Beckhoff_EPP2xxxEK1122.A_0059_EPP2339_0021_0017.WcState.InputToggle <-> WcState/InputToggle
//     PlcTask Inputs/GVL_iXlinker.EtherCAT_Master_EPPxxxx.Beckhoff_EPP2xxx.Beckhoff_EPP2xxxEK1122.A_0059_EPP2339_0021_0017.InfoData.State <-> InfoData/State
//   PLC/PLC Instance <-> EtherCAT Master EPPxxxx/Beckhoff EPP2xxx/Beckhoff EPP2xxxEK1122/A_0060(EPP2339-0021-0018)
//     PlcTask Inputs/GVL_iXlinker.EtherCAT_Master_EPPxxxx.Beckhoff_EPP2xxx.Beckhoff_EPP2xxxEK1122.A_0060_EPP2339_0021_0018.Channel_1.Input <-> Channel 1/Input
//     PlcTask Inputs/GVL_iXlinker.EtherCAT_Master_EPPxxxx.Beckhoff_EPP2xxx.Beckhoff_EPP2xxxEK1122.A_0060_EPP2339_0021_0018.Channel_2.Input <-> Channel 2/Input
//     PlcTask Inputs/GVL_iXlinker.EtherCAT_Master_EPPxxxx.Beckhoff_EPP2xxx.Beckhoff_EPP2xxxEK1122.A_0060_EPP2339_0021_0018.Channel_3.Input <-> Channel 3/Input
//     PlcTask Inputs/GVL_iXlinker.EtherCAT_Master_EPPxxxx.Beckhoff_EPP2xxx.Beckhoff_EPP2xxxEK1122.A_0060_EPP2339_0021_0018.Channel_4.Input <-> Channel 4/Input
//     PlcTask Inputs/GVL_iXlinker.EtherCAT_Master_EPPxxxx.Beckhoff_EPP2xxx.Beckhoff_EPP2xxxEK1122.A_0060_EPP2339_0021_0018.Channel_5.Input <-> Channel 5/Input
//     PlcTask Inputs/GVL_iXlinker.EtherCAT_Master_EPPxxxx.Beckhoff_EPP2xxx.Beckhoff_EPP2xxxEK1122.A_0060_EPP2339_0021_0018.Channel_6.Input <-> Channel 6/Input
//     PlcTask Inputs/GVL_iXlinker.EtherCAT_Master_EPPxxxx.Beckhoff_EPP2xxx.Beckhoff_EPP2xxxEK1122.A_0060_EPP2339_0021_0018.Channel_7.Input <-> Channel 7/Input
//     PlcTask Inputs/GVL_iXlinker.EtherCAT_Master_EPPxxxx.Beckhoff_EPP2xxx.Beckhoff_EPP2xxxEK1122.A_0060_EPP2339_0021_0018.Channel_8.Input <-> Channel 8/Input
//     PlcTask Inputs/GVL_iXlinker.EtherCAT_Master_EPPxxxx.Beckhoff_EPP2xxx.Beckhoff_EPP2xxxEK1122.A_0060_EPP2339_0021_0018.Channel_9.Input <-> Channel 9/Input
//     PlcTask Inputs/GVL_iXlinker.EtherCAT_Master_EPPxxxx.Beckhoff_EPP2xxx.Beckhoff_EPP2xxxEK1122.A_0060_EPP2339_0021_0018.Channel_10.Input <-> Channel 10/Input
//     PlcTask Inputs/GVL_iXlinker.EtherCAT_Master_EPPxxxx.Beckhoff_EPP2xxx.Beckhoff_EPP2xxxEK1122.A_0060_EPP2339_0021_0018.Channel_11.Input <-> Channel 11/Input
//     PlcTask Inputs/GVL_iXlinker.EtherCAT_Master_EPPxxxx.Beckhoff_EPP2xxx.Beckhoff_EPP2xxxEK1122.A_0060_EPP2339_0021_0018.Channel_12.Input <-> Channel 12/Input
//     PlcTask Inputs/GVL_iXlinker.EtherCAT_Master_EPPxxxx.Beckhoff_EPP2xxx.Beckhoff_EPP2xxxEK1122.A_0060_EPP2339_0021_0018.Channel_13.Input <-> Channel 13/Input
//     PlcTask Inputs/GVL_iXlinker.EtherCAT_Master_EPPxxxx.Beckhoff_EPP2xxx.Beckhoff_EPP2xxxEK1122.A_0060_EPP2339_0021_0018.Channel_14.Input <-> Channel 14/Input
//     PlcTask Inputs/GVL_iXlinker.EtherCAT_Master_EPPxxxx.Beckhoff_EPP2xxx.Beckhoff_EPP2xxxEK1122.A_0060_EPP2339_0021_0018.Channel_15.Input <-> Channel 15/Input
//     PlcTask Inputs/GVL_iXlinker.EtherCAT_Master_EPPxxxx.Beckhoff_EPP2xxx.Beckhoff_EPP2xxxEK1122.A_0060_EPP2339_0021_0018.Channel_16.Input <-> Channel 16/Input
//     PlcTask Outputs/GVL_iXlinker.EtherCAT_Master_EPPxxxx.Beckhoff_EPP2xxx.Beckhoff_EPP2xxxEK1122.A_0060_EPP2339_0021_0018.Channel_17.Output <-> Channel 17/Output
//     PlcTask Outputs/GVL_iXlinker.EtherCAT_Master_EPPxxxx.Beckhoff_EPP2xxx.Beckhoff_EPP2xxxEK1122.A_0060_EPP2339_0021_0018.Channel_18.Output <-> Channel 18/Output
//     PlcTask Outputs/GVL_iXlinker.EtherCAT_Master_EPPxxxx.Beckhoff_EPP2xxx.Beckhoff_EPP2xxxEK1122.A_0060_EPP2339_0021_0018.Channel_19.Output <-> Channel 19/Output
//     PlcTask Outputs/GVL_iXlinker.EtherCAT_Master_EPPxxxx.Beckhoff_EPP2xxx.Beckhoff_EPP2xxxEK1122.A_0060_EPP2339_0021_0018.Channel_20.Output <-> Channel 20/Output
//     PlcTask Outputs/GVL_iXlinker.EtherCAT_Master_EPPxxxx.Beckhoff_EPP2xxx.Beckhoff_EPP2xxxEK1122.A_0060_EPP2339_0021_0018.Channel_21.Output <-> Channel 21/Output
//     PlcTask Outputs/GVL_iXlinker.EtherCAT_Master_EPPxxxx.Beckhoff_EPP2xxx.Beckhoff_EPP2xxxEK1122.A_0060_EPP2339_0021_0018.Channel_22.Output <-> Channel 22/Output
//     PlcTask Outputs/GVL_iXlinker.EtherCAT_Master_EPPxxxx.Beckhoff_EPP2xxx.Beckhoff_EPP2xxxEK1122.A_0060_EPP2339_0021_0018.Channel_23.Output <-> Channel 23/Output
//     PlcTask Outputs/GVL_iXlinker.EtherCAT_Master_EPPxxxx.Beckhoff_EPP2xxx.Beckhoff_EPP2xxxEK1122.A_0060_EPP2339_0021_0018.Channel_24.Output <-> Channel 24/Output
//     PlcTask Outputs/GVL_iXlinker.EtherCAT_Master_EPPxxxx.Beckhoff_EPP2xxx.Beckhoff_EPP2xxxEK1122.A_0060_EPP2339_0021_0018.Channel_25.Output <-> Channel 25/Output
//     PlcTask Outputs/GVL_iXlinker.EtherCAT_Master_EPPxxxx.Beckhoff_EPP2xxx.Beckhoff_EPP2xxxEK1122.A_0060_EPP2339_0021_0018.Channel_26.Output <-> Channel 26/Output
//     PlcTask Outputs/GVL_iXlinker.EtherCAT_Master_EPPxxxx.Beckhoff_EPP2xxx.Beckhoff_EPP2xxxEK1122.A_0060_EPP2339_0021_0018.Channel_27.Output <-> Channel 27/Output
//     PlcTask Outputs/GVL_iXlinker.EtherCAT_Master_EPPxxxx.Beckhoff_EPP2xxx.Beckhoff_EPP2xxxEK1122.A_0060_EPP2339_0021_0018.Channel_28.Output <-> Channel 28/Output
//     PlcTask Outputs/GVL_iXlinker.EtherCAT_Master_EPPxxxx.Beckhoff_EPP2xxx.Beckhoff_EPP2xxxEK1122.A_0060_EPP2339_0021_0018.Channel_29.Output <-> Channel 29/Output
//     PlcTask Outputs/GVL_iXlinker.EtherCAT_Master_EPPxxxx.Beckhoff_EPP2xxx.Beckhoff_EPP2xxxEK1122.A_0060_EPP2339_0021_0018.Channel_30.Output <-> Channel 30/Output
//     PlcTask Outputs/GVL_iXlinker.EtherCAT_Master_EPPxxxx.Beckhoff_EPP2xxx.Beckhoff_EPP2xxxEK1122.A_0060_EPP2339_0021_0018.Channel_31.Output <-> Channel 31/Output
//     PlcTask Outputs/GVL_iXlinker.EtherCAT_Master_EPPxxxx.Beckhoff_EPP2xxx.Beckhoff_EPP2xxxEK1122.A_0060_EPP2339_0021_0018.Channel_32.Output <-> Channel 32/Output
//     PlcTask Inputs/GVL_iXlinker.EtherCAT_Master_EPPxxxx.Beckhoff_EPP2xxx.Beckhoff_EPP2xxxEK1122.A_0060_EPP2339_0021_0018.WcState.WcState <-> WcState/WcState
//     PlcTask Inputs/GVL_iXlinker.EtherCAT_Master_EPPxxxx.Beckhoff_EPP2xxx.Beckhoff_EPP2xxxEK1122.A_0060_EPP2339_0021_0018.WcState.InputToggle <-> WcState/InputToggle
//     PlcTask Inputs/GVL_iXlinker.EtherCAT_Master_EPPxxxx.Beckhoff_EPP2xxx.Beckhoff_EPP2xxxEK1122.A_0060_EPP2339_0021_0018.InfoData.State <-> InfoData/State
//   PLC/PLC Instance <-> EtherCAT Master EPPxxxx/Beckhoff EPP2xxx/Beckhoff EPP2xxxEK1122/A_0061(EPP2339-0022-0016)
//     PlcTask Inputs/GVL_iXlinker.EtherCAT_Master_EPPxxxx.Beckhoff_EPP2xxx.Beckhoff_EPP2xxxEK1122.A_0061_EPP2339_0022_0016.Channel_1.Input <-> Channel 1/Input
//     PlcTask Inputs/GVL_iXlinker.EtherCAT_Master_EPPxxxx.Beckhoff_EPP2xxx.Beckhoff_EPP2xxxEK1122.A_0061_EPP2339_0022_0016.Channel_2.Input <-> Channel 2/Input
//     PlcTask Inputs/GVL_iXlinker.EtherCAT_Master_EPPxxxx.Beckhoff_EPP2xxx.Beckhoff_EPP2xxxEK1122.A_0061_EPP2339_0022_0016.Channel_3.Input <-> Channel 3/Input
//     PlcTask Inputs/GVL_iXlinker.EtherCAT_Master_EPPxxxx.Beckhoff_EPP2xxx.Beckhoff_EPP2xxxEK1122.A_0061_EPP2339_0022_0016.Channel_4.Input <-> Channel 4/Input
//     PlcTask Inputs/GVL_iXlinker.EtherCAT_Master_EPPxxxx.Beckhoff_EPP2xxx.Beckhoff_EPP2xxxEK1122.A_0061_EPP2339_0022_0016.Channel_5.Input <-> Channel 5/Input
//     PlcTask Inputs/GVL_iXlinker.EtherCAT_Master_EPPxxxx.Beckhoff_EPP2xxx.Beckhoff_EPP2xxxEK1122.A_0061_EPP2339_0022_0016.Channel_6.Input <-> Channel 6/Input
//     PlcTask Inputs/GVL_iXlinker.EtherCAT_Master_EPPxxxx.Beckhoff_EPP2xxx.Beckhoff_EPP2xxxEK1122.A_0061_EPP2339_0022_0016.Channel_7.Input <-> Channel 7/Input
//     PlcTask Inputs/GVL_iXlinker.EtherCAT_Master_EPPxxxx.Beckhoff_EPP2xxx.Beckhoff_EPP2xxxEK1122.A_0061_EPP2339_0022_0016.Channel_8.Input <-> Channel 8/Input
//     PlcTask Inputs/GVL_iXlinker.EtherCAT_Master_EPPxxxx.Beckhoff_EPP2xxx.Beckhoff_EPP2xxxEK1122.A_0061_EPP2339_0022_0016.Channel_9.Input <-> Channel 9/Input
//     PlcTask Inputs/GVL_iXlinker.EtherCAT_Master_EPPxxxx.Beckhoff_EPP2xxx.Beckhoff_EPP2xxxEK1122.A_0061_EPP2339_0022_0016.Channel_10.Input <-> Channel 10/Input
//     PlcTask Inputs/GVL_iXlinker.EtherCAT_Master_EPPxxxx.Beckhoff_EPP2xxx.Beckhoff_EPP2xxxEK1122.A_0061_EPP2339_0022_0016.Channel_11.Input <-> Channel 11/Input
//     PlcTask Inputs/GVL_iXlinker.EtherCAT_Master_EPPxxxx.Beckhoff_EPP2xxx.Beckhoff_EPP2xxxEK1122.A_0061_EPP2339_0022_0016.Channel_12.Input <-> Channel 12/Input
//     PlcTask Inputs/GVL_iXlinker.EtherCAT_Master_EPPxxxx.Beckhoff_EPP2xxx.Beckhoff_EPP2xxxEK1122.A_0061_EPP2339_0022_0016.Channel_13.Input <-> Channel 13/Input
//     PlcTask Inputs/GVL_iXlinker.EtherCAT_Master_EPPxxxx.Beckhoff_EPP2xxx.Beckhoff_EPP2xxxEK1122.A_0061_EPP2339_0022_0016.Channel_14.Input <-> Channel 14/Input
//     PlcTask Inputs/GVL_iXlinker.EtherCAT_Master_EPPxxxx.Beckhoff_EPP2xxx.Beckhoff_EPP2xxxEK1122.A_0061_EPP2339_0022_0016.Channel_15.Input <-> Channel 15/Input
//     PlcTask Inputs/GVL_iXlinker.EtherCAT_Master_EPPxxxx.Beckhoff_EPP2xxx.Beckhoff_EPP2xxxEK1122.A_0061_EPP2339_0022_0016.Channel_16.Input <-> Channel 16/Input
//     PlcTask Outputs/GVL_iXlinker.EtherCAT_Master_EPPxxxx.Beckhoff_EPP2xxx.Beckhoff_EPP2xxxEK1122.A_0061_EPP2339_0022_0016.Channel_9_1.Output <-> Channel 9_1/Output
//     PlcTask Outputs/GVL_iXlinker.EtherCAT_Master_EPPxxxx.Beckhoff_EPP2xxx.Beckhoff_EPP2xxxEK1122.A_0061_EPP2339_0022_0016.Channel_10_1.Output <-> Channel 10_1/Output
//     PlcTask Outputs/GVL_iXlinker.EtherCAT_Master_EPPxxxx.Beckhoff_EPP2xxx.Beckhoff_EPP2xxxEK1122.A_0061_EPP2339_0022_0016.Channel_11_1.Output <-> Channel 11_1/Output
//     PlcTask Outputs/GVL_iXlinker.EtherCAT_Master_EPPxxxx.Beckhoff_EPP2xxx.Beckhoff_EPP2xxxEK1122.A_0061_EPP2339_0022_0016.Channel_12_1.Output <-> Channel 12_1/Output
//     PlcTask Outputs/GVL_iXlinker.EtherCAT_Master_EPPxxxx.Beckhoff_EPP2xxx.Beckhoff_EPP2xxxEK1122.A_0061_EPP2339_0022_0016.Channel_13_1.Output <-> Channel 13_1/Output
//     PlcTask Outputs/GVL_iXlinker.EtherCAT_Master_EPPxxxx.Beckhoff_EPP2xxx.Beckhoff_EPP2xxxEK1122.A_0061_EPP2339_0022_0016.Channel_14_1.Output <-> Channel 14_1/Output
//     PlcTask Outputs/GVL_iXlinker.EtherCAT_Master_EPPxxxx.Beckhoff_EPP2xxx.Beckhoff_EPP2xxxEK1122.A_0061_EPP2339_0022_0016.Channel_15_1.Output <-> Channel 15_1/Output
//     PlcTask Outputs/GVL_iXlinker.EtherCAT_Master_EPPxxxx.Beckhoff_EPP2xxx.Beckhoff_EPP2xxxEK1122.A_0061_EPP2339_0022_0016.Channel_16_1.Output <-> Channel 16_1/Output
//     PlcTask Outputs/GVL_iXlinker.EtherCAT_Master_EPPxxxx.Beckhoff_EPP2xxx.Beckhoff_EPP2xxxEK1122.A_0061_EPP2339_0022_0016.Channel_25.Output <-> Channel 25/Output
//     PlcTask Outputs/GVL_iXlinker.EtherCAT_Master_EPPxxxx.Beckhoff_EPP2xxx.Beckhoff_EPP2xxxEK1122.A_0061_EPP2339_0022_0016.Channel_26.Output <-> Channel 26/Output
//     PlcTask Outputs/GVL_iXlinker.EtherCAT_Master_EPPxxxx.Beckhoff_EPP2xxx.Beckhoff_EPP2xxxEK1122.A_0061_EPP2339_0022_0016.Channel_27.Output <-> Channel 27/Output
//     PlcTask Outputs/GVL_iXlinker.EtherCAT_Master_EPPxxxx.Beckhoff_EPP2xxx.Beckhoff_EPP2xxxEK1122.A_0061_EPP2339_0022_0016.Channel_28.Output <-> Channel 28/Output
//     PlcTask Outputs/GVL_iXlinker.EtherCAT_Master_EPPxxxx.Beckhoff_EPP2xxx.Beckhoff_EPP2xxxEK1122.A_0061_EPP2339_0022_0016.Channel_29.Output <-> Channel 29/Output
//     PlcTask Outputs/GVL_iXlinker.EtherCAT_Master_EPPxxxx.Beckhoff_EPP2xxx.Beckhoff_EPP2xxxEK1122.A_0061_EPP2339_0022_0016.Channel_30.Output <-> Channel 30/Output
//     PlcTask Outputs/GVL_iXlinker.EtherCAT_Master_EPPxxxx.Beckhoff_EPP2xxx.Beckhoff_EPP2xxxEK1122.A_0061_EPP2339_0022_0016.Channel_31.Output <-> Channel 31/Output
//     PlcTask Outputs/GVL_iXlinker.EtherCAT_Master_EPPxxxx.Beckhoff_EPP2xxx.Beckhoff_EPP2xxxEK1122.A_0061_EPP2339_0022_0016.Channel_32.Output <-> Channel 32/Output
//     PlcTask Inputs/GVL_iXlinker.EtherCAT_Master_EPPxxxx.Beckhoff_EPP2xxx.Beckhoff_EPP2xxxEK1122.A_0061_EPP2339_0022_0016.WcState.WcState <-> WcState/WcState
//     PlcTask Inputs/GVL_iXlinker.EtherCAT_Master_EPPxxxx.Beckhoff_EPP2xxx.Beckhoff_EPP2xxxEK1122.A_0061_EPP2339_0022_0016.WcState.InputToggle <-> WcState/InputToggle
//     PlcTask Inputs/GVL_iXlinker.EtherCAT_Master_EPPxxxx.Beckhoff_EPP2xxx.Beckhoff_EPP2xxxEK1122.A_0061_EPP2339_0022_0016.InfoData.State <-> InfoData/State
//   PLC/PLC Instance <-> EtherCAT Master EPPxxxx/Beckhoff EPP2xxx/Beckhoff EPP2xxxEK1122/A_0062(EPP2339-0022-0017)
//     PlcTask Inputs/GVL_iXlinker.EtherCAT_Master_EPPxxxx.Beckhoff_EPP2xxx.Beckhoff_EPP2xxxEK1122.A_0062_EPP2339_0022_0017.Channel_1.Input <-> Channel 1/Input
//     PlcTask Inputs/GVL_iXlinker.EtherCAT_Master_EPPxxxx.Beckhoff_EPP2xxx.Beckhoff_EPP2xxxEK1122.A_0062_EPP2339_0022_0017.Channel_2.Input <-> Channel 2/Input
//     PlcTask Inputs/GVL_iXlinker.EtherCAT_Master_EPPxxxx.Beckhoff_EPP2xxx.Beckhoff_EPP2xxxEK1122.A_0062_EPP2339_0022_0017.Channel_3.Input <-> Channel 3/Input
//     PlcTask Inputs/GVL_iXlinker.EtherCAT_Master_EPPxxxx.Beckhoff_EPP2xxx.Beckhoff_EPP2xxxEK1122.A_0062_EPP2339_0022_0017.Channel_4.Input <-> Channel 4/Input
//     PlcTask Inputs/GVL_iXlinker.EtherCAT_Master_EPPxxxx.Beckhoff_EPP2xxx.Beckhoff_EPP2xxxEK1122.A_0062_EPP2339_0022_0017.Channel_5.Input <-> Channel 5/Input
//     PlcTask Inputs/GVL_iXlinker.EtherCAT_Master_EPPxxxx.Beckhoff_EPP2xxx.Beckhoff_EPP2xxxEK1122.A_0062_EPP2339_0022_0017.Channel_6.Input <-> Channel 6/Input
//     PlcTask Inputs/GVL_iXlinker.EtherCAT_Master_EPPxxxx.Beckhoff_EPP2xxx.Beckhoff_EPP2xxxEK1122.A_0062_EPP2339_0022_0017.Channel_7.Input <-> Channel 7/Input
//     PlcTask Inputs/GVL_iXlinker.EtherCAT_Master_EPPxxxx.Beckhoff_EPP2xxx.Beckhoff_EPP2xxxEK1122.A_0062_EPP2339_0022_0017.Channel_8.Input <-> Channel 8/Input
//     PlcTask Inputs/GVL_iXlinker.EtherCAT_Master_EPPxxxx.Beckhoff_EPP2xxx.Beckhoff_EPP2xxxEK1122.A_0062_EPP2339_0022_0017.Channel_9.Input <-> Channel 9/Input
//     PlcTask Inputs/GVL_iXlinker.EtherCAT_Master_EPPxxxx.Beckhoff_EPP2xxx.Beckhoff_EPP2xxxEK1122.A_0062_EPP2339_0022_0017.Channel_10.Input <-> Channel 10/Input
//     PlcTask Inputs/GVL_iXlinker.EtherCAT_Master_EPPxxxx.Beckhoff_EPP2xxx.Beckhoff_EPP2xxxEK1122.A_0062_EPP2339_0022_0017.Channel_11.Input <-> Channel 11/Input
//     PlcTask Inputs/GVL_iXlinker.EtherCAT_Master_EPPxxxx.Beckhoff_EPP2xxx.Beckhoff_EPP2xxxEK1122.A_0062_EPP2339_0022_0017.Channel_12.Input <-> Channel 12/Input
//     PlcTask Inputs/GVL_iXlinker.EtherCAT_Master_EPPxxxx.Beckhoff_EPP2xxx.Beckhoff_EPP2xxxEK1122.A_0062_EPP2339_0022_0017.Channel_13.Input <-> Channel 13/Input
//     PlcTask Inputs/GVL_iXlinker.EtherCAT_Master_EPPxxxx.Beckhoff_EPP2xxx.Beckhoff_EPP2xxxEK1122.A_0062_EPP2339_0022_0017.Channel_14.Input <-> Channel 14/Input
//     PlcTask Inputs/GVL_iXlinker.EtherCAT_Master_EPPxxxx.Beckhoff_EPP2xxx.Beckhoff_EPP2xxxEK1122.A_0062_EPP2339_0022_0017.Channel_15.Input <-> Channel 15/Input
//     PlcTask Inputs/GVL_iXlinker.EtherCAT_Master_EPPxxxx.Beckhoff_EPP2xxx.Beckhoff_EPP2xxxEK1122.A_0062_EPP2339_0022_0017.Channel_16.Input <-> Channel 16/Input
//     PlcTask Outputs/GVL_iXlinker.EtherCAT_Master_EPPxxxx.Beckhoff_EPP2xxx.Beckhoff_EPP2xxxEK1122.A_0062_EPP2339_0022_0017.Channel_17.Output <-> Channel 17/Output
//     PlcTask Outputs/GVL_iXlinker.EtherCAT_Master_EPPxxxx.Beckhoff_EPP2xxx.Beckhoff_EPP2xxxEK1122.A_0062_EPP2339_0022_0017.Channel_18.Output <-> Channel 18/Output
//     PlcTask Outputs/GVL_iXlinker.EtherCAT_Master_EPPxxxx.Beckhoff_EPP2xxx.Beckhoff_EPP2xxxEK1122.A_0062_EPP2339_0022_0017.Channel_19.Output <-> Channel 19/Output
//     PlcTask Outputs/GVL_iXlinker.EtherCAT_Master_EPPxxxx.Beckhoff_EPP2xxx.Beckhoff_EPP2xxxEK1122.A_0062_EPP2339_0022_0017.Channel_20.Output <-> Channel 20/Output
//     PlcTask Outputs/GVL_iXlinker.EtherCAT_Master_EPPxxxx.Beckhoff_EPP2xxx.Beckhoff_EPP2xxxEK1122.A_0062_EPP2339_0022_0017.Channel_21.Output <-> Channel 21/Output
//     PlcTask Outputs/GVL_iXlinker.EtherCAT_Master_EPPxxxx.Beckhoff_EPP2xxx.Beckhoff_EPP2xxxEK1122.A_0062_EPP2339_0022_0017.Channel_22.Output <-> Channel 22/Output
//     PlcTask Outputs/GVL_iXlinker.EtherCAT_Master_EPPxxxx.Beckhoff_EPP2xxx.Beckhoff_EPP2xxxEK1122.A_0062_EPP2339_0022_0017.Channel_23.Output <-> Channel 23/Output
//     PlcTask Outputs/GVL_iXlinker.EtherCAT_Master_EPPxxxx.Beckhoff_EPP2xxx.Beckhoff_EPP2xxxEK1122.A_0062_EPP2339_0022_0017.Channel_24.Output <-> Channel 24/Output
//     PlcTask Outputs/GVL_iXlinker.EtherCAT_Master_EPPxxxx.Beckhoff_EPP2xxx.Beckhoff_EPP2xxxEK1122.A_0062_EPP2339_0022_0017.Channel_25.Output <-> Channel 25/Output
//     PlcTask Outputs/GVL_iXlinker.EtherCAT_Master_EPPxxxx.Beckhoff_EPP2xxx.Beckhoff_EPP2xxxEK1122.A_0062_EPP2339_0022_0017.Channel_26.Output <-> Channel 26/Output
//     PlcTask Outputs/GVL_iXlinker.EtherCAT_Master_EPPxxxx.Beckhoff_EPP2xxx.Beckhoff_EPP2xxxEK1122.A_0062_EPP2339_0022_0017.Channel_27.Output <-> Channel 27/Output
//     PlcTask Outputs/GVL_iXlinker.EtherCAT_Master_EPPxxxx.Beckhoff_EPP2xxx.Beckhoff_EPP2xxxEK1122.A_0062_EPP2339_0022_0017.Channel_28.Output <-> Channel 28/Output
//     PlcTask Outputs/GVL_iXlinker.EtherCAT_Master_EPPxxxx.Beckhoff_EPP2xxx.Beckhoff_EPP2xxxEK1122.A_0062_EPP2339_0022_0017.Channel_29.Output <-> Channel 29/Output
//     PlcTask Outputs/GVL_iXlinker.EtherCAT_Master_EPPxxxx.Beckhoff_EPP2xxx.Beckhoff_EPP2xxxEK1122.A_0062_EPP2339_0022_0017.Channel_30.Output <-> Channel 30/Output
//     PlcTask Outputs/GVL_iXlinker.EtherCAT_Master_EPPxxxx.Beckhoff_EPP2xxx.Beckhoff_EPP2xxxEK1122.A_0062_EPP2339_0022_0017.Channel_31.Output <-> Channel 31/Output
//     PlcTask Outputs/GVL_iXlinker.EtherCAT_Master_EPPxxxx.Beckhoff_EPP2xxx.Beckhoff_EPP2xxxEK1122.A_0062_EPP2339_0022_0017.Channel_32.Output <-> Channel 32/Output
//     PlcTask Inputs/GVL_iXlinker.EtherCAT_Master_EPPxxxx.Beckhoff_EPP2xxx.Beckhoff_EPP2xxxEK1122.A_0062_EPP2339_0022_0017.WcState.WcState <-> WcState/WcState
//     PlcTask Inputs/GVL_iXlinker.EtherCAT_Master_EPPxxxx.Beckhoff_EPP2xxx.Beckhoff_EPP2xxxEK1122.A_0062_EPP2339_0022_0017.WcState.InputToggle <-> WcState/InputToggle
//     PlcTask Inputs/GVL_iXlinker.EtherCAT_Master_EPPxxxx.Beckhoff_EPP2xxx.Beckhoff_EPP2xxxEK1122.A_0062_EPP2339_0022_0017.InfoData.State <-> InfoData/State
//   PLC/PLC Instance <-> EtherCAT Master EPPxxxx/Beckhoff EPP2xxx/Beckhoff EPP2xxxEK1122/A_0063(EPP2339-0022-0018)
//     PlcTask Inputs/GVL_iXlinker.EtherCAT_Master_EPPxxxx.Beckhoff_EPP2xxx.Beckhoff_EPP2xxxEK1122.A_0063_EPP2339_0022_0018.Channel_1.Input <-> Channel 1/Input
//     PlcTask Inputs/GVL_iXlinker.EtherCAT_Master_EPPxxxx.Beckhoff_EPP2xxx.Beckhoff_EPP2xxxEK1122.A_0063_EPP2339_0022_0018.Channel_2.Input <-> Channel 2/Input
//     PlcTask Inputs/GVL_iXlinker.EtherCAT_Master_EPPxxxx.Beckhoff_EPP2xxx.Beckhoff_EPP2xxxEK1122.A_0063_EPP2339_0022_0018.Channel_3.Input <-> Channel 3/Input
//     PlcTask Inputs/GVL_iXlinker.EtherCAT_Master_EPPxxxx.Beckhoff_EPP2xxx.Beckhoff_EPP2xxxEK1122.A_0063_EPP2339_0022_0018.Channel_4.Input <-> Channel 4/Input
//     PlcTask Inputs/GVL_iXlinker.EtherCAT_Master_EPPxxxx.Beckhoff_EPP2xxx.Beckhoff_EPP2xxxEK1122.A_0063_EPP2339_0022_0018.Channel_5.Input <-> Channel 5/Input
//     PlcTask Inputs/GVL_iXlinker.EtherCAT_Master_EPPxxxx.Beckhoff_EPP2xxx.Beckhoff_EPP2xxxEK1122.A_0063_EPP2339_0022_0018.Channel_6.Input <-> Channel 6/Input
//     PlcTask Inputs/GVL_iXlinker.EtherCAT_Master_EPPxxxx.Beckhoff_EPP2xxx.Beckhoff_EPP2xxxEK1122.A_0063_EPP2339_0022_0018.Channel_7.Input <-> Channel 7/Input
//     PlcTask Inputs/GVL_iXlinker.EtherCAT_Master_EPPxxxx.Beckhoff_EPP2xxx.Beckhoff_EPP2xxxEK1122.A_0063_EPP2339_0022_0018.Channel_8.Input <-> Channel 8/Input
//     PlcTask Inputs/GVL_iXlinker.EtherCAT_Master_EPPxxxx.Beckhoff_EPP2xxx.Beckhoff_EPP2xxxEK1122.A_0063_EPP2339_0022_0018.Channel_9.Input <-> Channel 9/Input
//     PlcTask Inputs/GVL_iXlinker.EtherCAT_Master_EPPxxxx.Beckhoff_EPP2xxx.Beckhoff_EPP2xxxEK1122.A_0063_EPP2339_0022_0018.Channel_10.Input <-> Channel 10/Input
//     PlcTask Inputs/GVL_iXlinker.EtherCAT_Master_EPPxxxx.Beckhoff_EPP2xxx.Beckhoff_EPP2xxxEK1122.A_0063_EPP2339_0022_0018.Channel_11.Input <-> Channel 11/Input
//     PlcTask Inputs/GVL_iXlinker.EtherCAT_Master_EPPxxxx.Beckhoff_EPP2xxx.Beckhoff_EPP2xxxEK1122.A_0063_EPP2339_0022_0018.Channel_12.Input <-> Channel 12/Input
//     PlcTask Inputs/GVL_iXlinker.EtherCAT_Master_EPPxxxx.Beckhoff_EPP2xxx.Beckhoff_EPP2xxxEK1122.A_0063_EPP2339_0022_0018.Channel_13.Input <-> Channel 13/Input
//     PlcTask Inputs/GVL_iXlinker.EtherCAT_Master_EPPxxxx.Beckhoff_EPP2xxx.Beckhoff_EPP2xxxEK1122.A_0063_EPP2339_0022_0018.Channel_14.Input <-> Channel 14/Input
//     PlcTask Inputs/GVL_iXlinker.EtherCAT_Master_EPPxxxx.Beckhoff_EPP2xxx.Beckhoff_EPP2xxxEK1122.A_0063_EPP2339_0022_0018.Channel_15.Input <-> Channel 15/Input
//     PlcTask Inputs/GVL_iXlinker.EtherCAT_Master_EPPxxxx.Beckhoff_EPP2xxx.Beckhoff_EPP2xxxEK1122.A_0063_EPP2339_0022_0018.Channel_16.Input <-> Channel 16/Input
//     PlcTask Outputs/GVL_iXlinker.EtherCAT_Master_EPPxxxx.Beckhoff_EPP2xxx.Beckhoff_EPP2xxxEK1122.A_0063_EPP2339_0022_0018.Channel_17.Output <-> Channel 17/Output
//     PlcTask Outputs/GVL_iXlinker.EtherCAT_Master_EPPxxxx.Beckhoff_EPP2xxx.Beckhoff_EPP2xxxEK1122.A_0063_EPP2339_0022_0018.Channel_18.Output <-> Channel 18/Output
//     PlcTask Outputs/GVL_iXlinker.EtherCAT_Master_EPPxxxx.Beckhoff_EPP2xxx.Beckhoff_EPP2xxxEK1122.A_0063_EPP2339_0022_0018.Channel_19.Output <-> Channel 19/Output
//     PlcTask Outputs/GVL_iXlinker.EtherCAT_Master_EPPxxxx.Beckhoff_EPP2xxx.Beckhoff_EPP2xxxEK1122.A_0063_EPP2339_0022_0018.Channel_20.Output <-> Channel 20/Output
//     PlcTask Outputs/GVL_iXlinker.EtherCAT_Master_EPPxxxx.Beckhoff_EPP2xxx.Beckhoff_EPP2xxxEK1122.A_0063_EPP2339_0022_0018.Channel_21.Output <-> Channel 21/Output
//     PlcTask Outputs/GVL_iXlinker.EtherCAT_Master_EPPxxxx.Beckhoff_EPP2xxx.Beckhoff_EPP2xxxEK1122.A_0063_EPP2339_0022_0018.Channel_22.Output <-> Channel 22/Output
//     PlcTask Outputs/GVL_iXlinker.EtherCAT_Master_EPPxxxx.Beckhoff_EPP2xxx.Beckhoff_EPP2xxxEK1122.A_0063_EPP2339_0022_0018.Channel_23.Output <-> Channel 23/Output
//     PlcTask Outputs/GVL_iXlinker.EtherCAT_Master_EPPxxxx.Beckhoff_EPP2xxx.Beckhoff_EPP2xxxEK1122.A_0063_EPP2339_0022_0018.Channel_24.Output <-> Channel 24/Output
//     PlcTask Outputs/GVL_iXlinker.EtherCAT_Master_EPPxxxx.Beckhoff_EPP2xxx.Beckhoff_EPP2xxxEK1122.A_0063_EPP2339_0022_0018.Channel_25.Output <-> Channel 25/Output
//     PlcTask Outputs/GVL_iXlinker.EtherCAT_Master_EPPxxxx.Beckhoff_EPP2xxx.Beckhoff_EPP2xxxEK1122.A_0063_EPP2339_0022_0018.Channel_26.Output <-> Channel 26/Output
//     PlcTask Outputs/GVL_iXlinker.EtherCAT_Master_EPPxxxx.Beckhoff_EPP2xxx.Beckhoff_EPP2xxxEK1122.A_0063_EPP2339_0022_0018.Channel_27.Output <-> Channel 27/Output
//     PlcTask Outputs/GVL_iXlinker.EtherCAT_Master_EPPxxxx.Beckhoff_EPP2xxx.Beckhoff_EPP2xxxEK1122.A_0063_EPP2339_0022_0018.Channel_28.Output <-> Channel 28/Output
//     PlcTask Outputs/GVL_iXlinker.EtherCAT_Master_EPPxxxx.Beckhoff_EPP2xxx.Beckhoff_EPP2xxxEK1122.A_0063_EPP2339_0022_0018.Channel_29.Output <-> Channel 29/Output
//     PlcTask Outputs/GVL_iXlinker.EtherCAT_Master_EPPxxxx.Beckhoff_EPP2xxx.Beckhoff_EPP2xxxEK1122.A_0063_EPP2339_0022_0018.Channel_30.Output <-> Channel 30/Output
//     PlcTask Outputs/GVL_iXlinker.EtherCAT_Master_EPPxxxx.Beckhoff_EPP2xxx.Beckhoff_EPP2xxxEK1122.A_0063_EPP2339_0022_0018.Channel_31.Output <-> Channel 31/Output
//     PlcTask Outputs/GVL_iXlinker.EtherCAT_Master_EPPxxxx.Beckhoff_EPP2xxx.Beckhoff_EPP2xxxEK1122.A_0063_EPP2339_0022_0018.Channel_32.Output <-> Channel 32/Output
//     PlcTask Inputs/GVL_iXlinker.EtherCAT_Master_EPPxxxx.Beckhoff_EPP2xxx.Beckhoff_EPP2xxxEK1122.A_0063_EPP2339_0022_0018.WcState.WcState <-> WcState/WcState
//     PlcTask Inputs/GVL_iXlinker.EtherCAT_Master_EPPxxxx.Beckhoff_EPP2xxx.Beckhoff_EPP2xxxEK1122.A_0063_EPP2339_0022_0018.WcState.InputToggle <-> WcState/InputToggle
//     PlcTask Inputs/GVL_iXlinker.EtherCAT_Master_EPPxxxx.Beckhoff_EPP2xxx.Beckhoff_EPP2xxxEK1122.A_0063_EPP2339_0022_0018.InfoData.State <-> InfoData/State
//   PLC/PLC Instance <-> EtherCAT Master EPPxxxx/Beckhoff EPP2xxx/Beckhoff EPP2xxxEK1122/A_0064(EPP2349-0021-0016)
//     PlcTask Inputs/GVL_iXlinker.EtherCAT_Master_EPPxxxx.Beckhoff_EPP2xxx.Beckhoff_EPP2xxxEK1122.A_0064_EPP2349_0021_0016.Channel_1.Input <-> Channel 1/Input
//     PlcTask Inputs/GVL_iXlinker.EtherCAT_Master_EPPxxxx.Beckhoff_EPP2xxx.Beckhoff_EPP2xxxEK1122.A_0064_EPP2349_0021_0016.Channel_2.Input <-> Channel 2/Input
//     PlcTask Inputs/GVL_iXlinker.EtherCAT_Master_EPPxxxx.Beckhoff_EPP2xxx.Beckhoff_EPP2xxxEK1122.A_0064_EPP2349_0021_0016.Channel_3.Input <-> Channel 3/Input
//     PlcTask Inputs/GVL_iXlinker.EtherCAT_Master_EPPxxxx.Beckhoff_EPP2xxx.Beckhoff_EPP2xxxEK1122.A_0064_EPP2349_0021_0016.Channel_4.Input <-> Channel 4/Input
//     PlcTask Inputs/GVL_iXlinker.EtherCAT_Master_EPPxxxx.Beckhoff_EPP2xxx.Beckhoff_EPP2xxxEK1122.A_0064_EPP2349_0021_0016.Channel_5.Input <-> Channel 5/Input
//     PlcTask Inputs/GVL_iXlinker.EtherCAT_Master_EPPxxxx.Beckhoff_EPP2xxx.Beckhoff_EPP2xxxEK1122.A_0064_EPP2349_0021_0016.Channel_6.Input <-> Channel 6/Input
//     PlcTask Inputs/GVL_iXlinker.EtherCAT_Master_EPPxxxx.Beckhoff_EPP2xxx.Beckhoff_EPP2xxxEK1122.A_0064_EPP2349_0021_0016.Channel_7.Input <-> Channel 7/Input
//     PlcTask Inputs/GVL_iXlinker.EtherCAT_Master_EPPxxxx.Beckhoff_EPP2xxx.Beckhoff_EPP2xxxEK1122.A_0064_EPP2349_0021_0016.Channel_8.Input <-> Channel 8/Input
//     PlcTask Inputs/GVL_iXlinker.EtherCAT_Master_EPPxxxx.Beckhoff_EPP2xxx.Beckhoff_EPP2xxxEK1122.A_0064_EPP2349_0021_0016.Channel_9.Input <-> Channel 9/Input
//     PlcTask Inputs/GVL_iXlinker.EtherCAT_Master_EPPxxxx.Beckhoff_EPP2xxx.Beckhoff_EPP2xxxEK1122.A_0064_EPP2349_0021_0016.Channel_10.Input <-> Channel 10/Input
//     PlcTask Inputs/GVL_iXlinker.EtherCAT_Master_EPPxxxx.Beckhoff_EPP2xxx.Beckhoff_EPP2xxxEK1122.A_0064_EPP2349_0021_0016.Channel_11.Input <-> Channel 11/Input
//     PlcTask Inputs/GVL_iXlinker.EtherCAT_Master_EPPxxxx.Beckhoff_EPP2xxx.Beckhoff_EPP2xxxEK1122.A_0064_EPP2349_0021_0016.Channel_12.Input <-> Channel 12/Input
//     PlcTask Inputs/GVL_iXlinker.EtherCAT_Master_EPPxxxx.Beckhoff_EPP2xxx.Beckhoff_EPP2xxxEK1122.A_0064_EPP2349_0021_0016.Channel_13.Input <-> Channel 13/Input
//     PlcTask Inputs/GVL_iXlinker.EtherCAT_Master_EPPxxxx.Beckhoff_EPP2xxx.Beckhoff_EPP2xxxEK1122.A_0064_EPP2349_0021_0016.Channel_14.Input <-> Channel 14/Input
//     PlcTask Inputs/GVL_iXlinker.EtherCAT_Master_EPPxxxx.Beckhoff_EPP2xxx.Beckhoff_EPP2xxxEK1122.A_0064_EPP2349_0021_0016.Channel_15.Input <-> Channel 15/Input
//     PlcTask Inputs/GVL_iXlinker.EtherCAT_Master_EPPxxxx.Beckhoff_EPP2xxx.Beckhoff_EPP2xxxEK1122.A_0064_EPP2349_0021_0016.Channel_16.Input <-> Channel 16/Input
//     PlcTask Outputs/GVL_iXlinker.EtherCAT_Master_EPPxxxx.Beckhoff_EPP2xxx.Beckhoff_EPP2xxxEK1122.A_0064_EPP2349_0021_0016.Channel_9_1.Output <-> Channel 9_1/Output
//     PlcTask Outputs/GVL_iXlinker.EtherCAT_Master_EPPxxxx.Beckhoff_EPP2xxx.Beckhoff_EPP2xxxEK1122.A_0064_EPP2349_0021_0016.Channel_10_1.Output <-> Channel 10_1/Output
//     PlcTask Outputs/GVL_iXlinker.EtherCAT_Master_EPPxxxx.Beckhoff_EPP2xxx.Beckhoff_EPP2xxxEK1122.A_0064_EPP2349_0021_0016.Channel_11_1.Output <-> Channel 11_1/Output
//     PlcTask Outputs/GVL_iXlinker.EtherCAT_Master_EPPxxxx.Beckhoff_EPP2xxx.Beckhoff_EPP2xxxEK1122.A_0064_EPP2349_0021_0016.Channel_12_1.Output <-> Channel 12_1/Output
//     PlcTask Outputs/GVL_iXlinker.EtherCAT_Master_EPPxxxx.Beckhoff_EPP2xxx.Beckhoff_EPP2xxxEK1122.A_0064_EPP2349_0021_0016.Channel_13_1.Output <-> Channel 13_1/Output
//     PlcTask Outputs/GVL_iXlinker.EtherCAT_Master_EPPxxxx.Beckhoff_EPP2xxx.Beckhoff_EPP2xxxEK1122.A_0064_EPP2349_0021_0016.Channel_14_1.Output <-> Channel 14_1/Output
//     PlcTask Outputs/GVL_iXlinker.EtherCAT_Master_EPPxxxx.Beckhoff_EPP2xxx.Beckhoff_EPP2xxxEK1122.A_0064_EPP2349_0021_0016.Channel_15_1.Output <-> Channel 15_1/Output
//     PlcTask Outputs/GVL_iXlinker.EtherCAT_Master_EPPxxxx.Beckhoff_EPP2xxx.Beckhoff_EPP2xxxEK1122.A_0064_EPP2349_0021_0016.Channel_16_1.Output <-> Channel 16_1/Output
//     PlcTask Outputs/GVL_iXlinker.EtherCAT_Master_EPPxxxx.Beckhoff_EPP2xxx.Beckhoff_EPP2xxxEK1122.A_0064_EPP2349_0021_0016.Channel_25.Output <-> Channel 25/Output
//     PlcTask Outputs/GVL_iXlinker.EtherCAT_Master_EPPxxxx.Beckhoff_EPP2xxx.Beckhoff_EPP2xxxEK1122.A_0064_EPP2349_0021_0016.Channel_26.Output <-> Channel 26/Output
//     PlcTask Outputs/GVL_iXlinker.EtherCAT_Master_EPPxxxx.Beckhoff_EPP2xxx.Beckhoff_EPP2xxxEK1122.A_0064_EPP2349_0021_0016.Channel_27.Output <-> Channel 27/Output
//     PlcTask Outputs/GVL_iXlinker.EtherCAT_Master_EPPxxxx.Beckhoff_EPP2xxx.Beckhoff_EPP2xxxEK1122.A_0064_EPP2349_0021_0016.Channel_28.Output <-> Channel 28/Output
//     PlcTask Outputs/GVL_iXlinker.EtherCAT_Master_EPPxxxx.Beckhoff_EPP2xxx.Beckhoff_EPP2xxxEK1122.A_0064_EPP2349_0021_0016.Channel_29.Output <-> Channel 29/Output
//     PlcTask Outputs/GVL_iXlinker.EtherCAT_Master_EPPxxxx.Beckhoff_EPP2xxx.Beckhoff_EPP2xxxEK1122.A_0064_EPP2349_0021_0016.Channel_30.Output <-> Channel 30/Output
//     PlcTask Outputs/GVL_iXlinker.EtherCAT_Master_EPPxxxx.Beckhoff_EPP2xxx.Beckhoff_EPP2xxxEK1122.A_0064_EPP2349_0021_0016.Channel_31.Output <-> Channel 31/Output
//     PlcTask Outputs/GVL_iXlinker.EtherCAT_Master_EPPxxxx.Beckhoff_EPP2xxx.Beckhoff_EPP2xxxEK1122.A_0064_EPP2349_0021_0016.Channel_32.Output <-> Channel 32/Output
//     PlcTask Inputs/GVL_iXlinker.EtherCAT_Master_EPPxxxx.Beckhoff_EPP2xxx.Beckhoff_EPP2xxxEK1122.A_0064_EPP2349_0021_0016.WcState.WcState <-> WcState/WcState
//     PlcTask Inputs/GVL_iXlinker.EtherCAT_Master_EPPxxxx.Beckhoff_EPP2xxx.Beckhoff_EPP2xxxEK1122.A_0064_EPP2349_0021_0016.WcState.InputToggle <-> WcState/InputToggle
//     PlcTask Inputs/GVL_iXlinker.EtherCAT_Master_EPPxxxx.Beckhoff_EPP2xxx.Beckhoff_EPP2xxxEK1122.A_0064_EPP2349_0021_0016.InfoData.State <-> InfoData/State
//   PLC/PLC Instance <-> EtherCAT Master EPPxxxx/Beckhoff EPP2xxx/Beckhoff EPP2xxxEK1122/A_0065(EPP2349-0021-0017)
//     PlcTask Inputs/GVL_iXlinker.EtherCAT_Master_EPPxxxx.Beckhoff_EPP2xxx.Beckhoff_EPP2xxxEK1122.A_0065_EPP2349_0021_0017.Channel_1.Input <-> Channel 1/Input
//     PlcTask Inputs/GVL_iXlinker.EtherCAT_Master_EPPxxxx.Beckhoff_EPP2xxx.Beckhoff_EPP2xxxEK1122.A_0065_EPP2349_0021_0017.Channel_2.Input <-> Channel 2/Input
//     PlcTask Inputs/GVL_iXlinker.EtherCAT_Master_EPPxxxx.Beckhoff_EPP2xxx.Beckhoff_EPP2xxxEK1122.A_0065_EPP2349_0021_0017.Channel_3.Input <-> Channel 3/Input
//     PlcTask Inputs/GVL_iXlinker.EtherCAT_Master_EPPxxxx.Beckhoff_EPP2xxx.Beckhoff_EPP2xxxEK1122.A_0065_EPP2349_0021_0017.Channel_4.Input <-> Channel 4/Input
//     PlcTask Inputs/GVL_iXlinker.EtherCAT_Master_EPPxxxx.Beckhoff_EPP2xxx.Beckhoff_EPP2xxxEK1122.A_0065_EPP2349_0021_0017.Channel_5.Input <-> Channel 5/Input
//     PlcTask Inputs/GVL_iXlinker.EtherCAT_Master_EPPxxxx.Beckhoff_EPP2xxx.Beckhoff_EPP2xxxEK1122.A_0065_EPP2349_0021_0017.Channel_6.Input <-> Channel 6/Input
//     PlcTask Inputs/GVL_iXlinker.EtherCAT_Master_EPPxxxx.Beckhoff_EPP2xxx.Beckhoff_EPP2xxxEK1122.A_0065_EPP2349_0021_0017.Channel_7.Input <-> Channel 7/Input
//     PlcTask Inputs/GVL_iXlinker.EtherCAT_Master_EPPxxxx.Beckhoff_EPP2xxx.Beckhoff_EPP2xxxEK1122.A_0065_EPP2349_0021_0017.Channel_8.Input <-> Channel 8/Input
//     PlcTask Inputs/GVL_iXlinker.EtherCAT_Master_EPPxxxx.Beckhoff_EPP2xxx.Beckhoff_EPP2xxxEK1122.A_0065_EPP2349_0021_0017.Channel_9.Input <-> Channel 9/Input
//     PlcTask Inputs/GVL_iXlinker.EtherCAT_Master_EPPxxxx.Beckhoff_EPP2xxx.Beckhoff_EPP2xxxEK1122.A_0065_EPP2349_0021_0017.Channel_10.Input <-> Channel 10/Input
//     PlcTask Inputs/GVL_iXlinker.EtherCAT_Master_EPPxxxx.Beckhoff_EPP2xxx.Beckhoff_EPP2xxxEK1122.A_0065_EPP2349_0021_0017.Channel_11.Input <-> Channel 11/Input
//     PlcTask Inputs/GVL_iXlinker.EtherCAT_Master_EPPxxxx.Beckhoff_EPP2xxx.Beckhoff_EPP2xxxEK1122.A_0065_EPP2349_0021_0017.Channel_12.Input <-> Channel 12/Input
//     PlcTask Inputs/GVL_iXlinker.EtherCAT_Master_EPPxxxx.Beckhoff_EPP2xxx.Beckhoff_EPP2xxxEK1122.A_0065_EPP2349_0021_0017.Channel_13.Input <-> Channel 13/Input
//     PlcTask Inputs/GVL_iXlinker.EtherCAT_Master_EPPxxxx.Beckhoff_EPP2xxx.Beckhoff_EPP2xxxEK1122.A_0065_EPP2349_0021_0017.Channel_14.Input <-> Channel 14/Input
//     PlcTask Inputs/GVL_iXlinker.EtherCAT_Master_EPPxxxx.Beckhoff_EPP2xxx.Beckhoff_EPP2xxxEK1122.A_0065_EPP2349_0021_0017.Channel_15.Input <-> Channel 15/Input
//     PlcTask Inputs/GVL_iXlinker.EtherCAT_Master_EPPxxxx.Beckhoff_EPP2xxx.Beckhoff_EPP2xxxEK1122.A_0065_EPP2349_0021_0017.Channel_16.Input <-> Channel 16/Input
//     PlcTask Outputs/GVL_iXlinker.EtherCAT_Master_EPPxxxx.Beckhoff_EPP2xxx.Beckhoff_EPP2xxxEK1122.A_0065_EPP2349_0021_0017.Channel_17.Output <-> Channel 17/Output
//     PlcTask Outputs/GVL_iXlinker.EtherCAT_Master_EPPxxxx.Beckhoff_EPP2xxx.Beckhoff_EPP2xxxEK1122.A_0065_EPP2349_0021_0017.Channel_18.Output <-> Channel 18/Output
//     PlcTask Outputs/GVL_iXlinker.EtherCAT_Master_EPPxxxx.Beckhoff_EPP2xxx.Beckhoff_EPP2xxxEK1122.A_0065_EPP2349_0021_0017.Channel_19.Output <-> Channel 19/Output
//     PlcTask Outputs/GVL_iXlinker.EtherCAT_Master_EPPxxxx.Beckhoff_EPP2xxx.Beckhoff_EPP2xxxEK1122.A_0065_EPP2349_0021_0017.Channel_20.Output <-> Channel 20/Output
//     PlcTask Outputs/GVL_iXlinker.EtherCAT_Master_EPPxxxx.Beckhoff_EPP2xxx.Beckhoff_EPP2xxxEK1122.A_0065_EPP2349_0021_0017.Channel_21.Output <-> Channel 21/Output
//     PlcTask Outputs/GVL_iXlinker.EtherCAT_Master_EPPxxxx.Beckhoff_EPP2xxx.Beckhoff_EPP2xxxEK1122.A_0065_EPP2349_0021_0017.Channel_22.Output <-> Channel 22/Output
//     PlcTask Outputs/GVL_iXlinker.EtherCAT_Master_EPPxxxx.Beckhoff_EPP2xxx.Beckhoff_EPP2xxxEK1122.A_0065_EPP2349_0021_0017.Channel_23.Output <-> Channel 23/Output
//     PlcTask Outputs/GVL_iXlinker.EtherCAT_Master_EPPxxxx.Beckhoff_EPP2xxx.Beckhoff_EPP2xxxEK1122.A_0065_EPP2349_0021_0017.Channel_24.Output <-> Channel 24/Output
//     PlcTask Outputs/GVL_iXlinker.EtherCAT_Master_EPPxxxx.Beckhoff_EPP2xxx.Beckhoff_EPP2xxxEK1122.A_0065_EPP2349_0021_0017.Channel_25.Output <-> Channel 25/Output
//     PlcTask Outputs/GVL_iXlinker.EtherCAT_Master_EPPxxxx.Beckhoff_EPP2xxx.Beckhoff_EPP2xxxEK1122.A_0065_EPP2349_0021_0017.Channel_26.Output <-> Channel 26/Output
//     PlcTask Outputs/GVL_iXlinker.EtherCAT_Master_EPPxxxx.Beckhoff_EPP2xxx.Beckhoff_EPP2xxxEK1122.A_0065_EPP2349_0021_0017.Channel_27.Output <-> Channel 27/Output
//     PlcTask Outputs/GVL_iXlinker.EtherCAT_Master_EPPxxxx.Beckhoff_EPP2xxx.Beckhoff_EPP2xxxEK1122.A_0065_EPP2349_0021_0017.Channel_28.Output <-> Channel 28/Output
//     PlcTask Outputs/GVL_iXlinker.EtherCAT_Master_EPPxxxx.Beckhoff_EPP2xxx.Beckhoff_EPP2xxxEK1122.A_0065_EPP2349_0021_0017.Channel_29.Output <-> Channel 29/Output
//     PlcTask Outputs/GVL_iXlinker.EtherCAT_Master_EPPxxxx.Beckhoff_EPP2xxx.Beckhoff_EPP2xxxEK1122.A_0065_EPP2349_0021_0017.Channel_30.Output <-> Channel 30/Output
//     PlcTask Outputs/GVL_iXlinker.EtherCAT_Master_EPPxxxx.Beckhoff_EPP2xxx.Beckhoff_EPP2xxxEK1122.A_0065_EPP2349_0021_0017.Channel_31.Output <-> Channel 31/Output
//     PlcTask Outputs/GVL_iXlinker.EtherCAT_Master_EPPxxxx.Beckhoff_EPP2xxx.Beckhoff_EPP2xxxEK1122.A_0065_EPP2349_0021_0017.Channel_32.Output <-> Channel 32/Output
//     PlcTask Inputs/GVL_iXlinker.EtherCAT_Master_EPPxxxx.Beckhoff_EPP2xxx.Beckhoff_EPP2xxxEK1122.A_0065_EPP2349_0021_0017.WcState.WcState <-> WcState/WcState
//     PlcTask Inputs/GVL_iXlinker.EtherCAT_Master_EPPxxxx.Beckhoff_EPP2xxx.Beckhoff_EPP2xxxEK1122.A_0065_EPP2349_0021_0017.WcState.InputToggle <-> WcState/InputToggle
//     PlcTask Inputs/GVL_iXlinker.EtherCAT_Master_EPPxxxx.Beckhoff_EPP2xxx.Beckhoff_EPP2xxxEK1122.A_0065_EPP2349_0021_0017.InfoData.State <-> InfoData/State
//   PLC/PLC Instance <-> EtherCAT Master EPPxxxx/Beckhoff EPP2xxx/Beckhoff EPP2xxxEK1122/A_0066(EPP2349-0021-0018)
//     PlcTask Inputs/GVL_iXlinker.EtherCAT_Master_EPPxxxx.Beckhoff_EPP2xxx.Beckhoff_EPP2xxxEK1122.A_0066_EPP2349_0021_0018.Channel_1.Input <-> Channel 1/Input
//     PlcTask Inputs/GVL_iXlinker.EtherCAT_Master_EPPxxxx.Beckhoff_EPP2xxx.Beckhoff_EPP2xxxEK1122.A_0066_EPP2349_0021_0018.Channel_2.Input <-> Channel 2/Input
//     PlcTask Inputs/GVL_iXlinker.EtherCAT_Master_EPPxxxx.Beckhoff_EPP2xxx.Beckhoff_EPP2xxxEK1122.A_0066_EPP2349_0021_0018.Channel_3.Input <-> Channel 3/Input
//     PlcTask Inputs/GVL_iXlinker.EtherCAT_Master_EPPxxxx.Beckhoff_EPP2xxx.Beckhoff_EPP2xxxEK1122.A_0066_EPP2349_0021_0018.Channel_4.Input <-> Channel 4/Input
//     PlcTask Inputs/GVL_iXlinker.EtherCAT_Master_EPPxxxx.Beckhoff_EPP2xxx.Beckhoff_EPP2xxxEK1122.A_0066_EPP2349_0021_0018.Channel_5.Input <-> Channel 5/Input
//     PlcTask Inputs/GVL_iXlinker.EtherCAT_Master_EPPxxxx.Beckhoff_EPP2xxx.Beckhoff_EPP2xxxEK1122.A_0066_EPP2349_0021_0018.Channel_6.Input <-> Channel 6/Input
//     PlcTask Inputs/GVL_iXlinker.EtherCAT_Master_EPPxxxx.Beckhoff_EPP2xxx.Beckhoff_EPP2xxxEK1122.A_0066_EPP2349_0021_0018.Channel_7.Input <-> Channel 7/Input
//     PlcTask Inputs/GVL_iXlinker.EtherCAT_Master_EPPxxxx.Beckhoff_EPP2xxx.Beckhoff_EPP2xxxEK1122.A_0066_EPP2349_0021_0018.Channel_8.Input <-> Channel 8/Input
//     PlcTask Inputs/GVL_iXlinker.EtherCAT_Master_EPPxxxx.Beckhoff_EPP2xxx.Beckhoff_EPP2xxxEK1122.A_0066_EPP2349_0021_0018.Channel_9.Input <-> Channel 9/Input
//     PlcTask Inputs/GVL_iXlinker.EtherCAT_Master_EPPxxxx.Beckhoff_EPP2xxx.Beckhoff_EPP2xxxEK1122.A_0066_EPP2349_0021_0018.Channel_10.Input <-> Channel 10/Input
//     PlcTask Inputs/GVL_iXlinker.EtherCAT_Master_EPPxxxx.Beckhoff_EPP2xxx.Beckhoff_EPP2xxxEK1122.A_0066_EPP2349_0021_0018.Channel_11.Input <-> Channel 11/Input
//     PlcTask Inputs/GVL_iXlinker.EtherCAT_Master_EPPxxxx.Beckhoff_EPP2xxx.Beckhoff_EPP2xxxEK1122.A_0066_EPP2349_0021_0018.Channel_12.Input <-> Channel 12/Input
//     PlcTask Inputs/GVL_iXlinker.EtherCAT_Master_EPPxxxx.Beckhoff_EPP2xxx.Beckhoff_EPP2xxxEK1122.A_0066_EPP2349_0021_0018.Channel_13.Input <-> Channel 13/Input
//     PlcTask Inputs/GVL_iXlinker.EtherCAT_Master_EPPxxxx.Beckhoff_EPP2xxx.Beckhoff_EPP2xxxEK1122.A_0066_EPP2349_0021_0018.Channel_14.Input <-> Channel 14/Input
//     PlcTask Inputs/GVL_iXlinker.EtherCAT_Master_EPPxxxx.Beckhoff_EPP2xxx.Beckhoff_EPP2xxxEK1122.A_0066_EPP2349_0021_0018.Channel_15.Input <-> Channel 15/Input
//     PlcTask Inputs/GVL_iXlinker.EtherCAT_Master_EPPxxxx.Beckhoff_EPP2xxx.Beckhoff_EPP2xxxEK1122.A_0066_EPP2349_0021_0018.Channel_16.Input <-> Channel 16/Input
//     PlcTask Outputs/GVL_iXlinker.EtherCAT_Master_EPPxxxx.Beckhoff_EPP2xxx.Beckhoff_EPP2xxxEK1122.A_0066_EPP2349_0021_0018.Channel_17.Output <-> Channel 17/Output
//     PlcTask Outputs/GVL_iXlinker.EtherCAT_Master_EPPxxxx.Beckhoff_EPP2xxx.Beckhoff_EPP2xxxEK1122.A_0066_EPP2349_0021_0018.Channel_18.Output <-> Channel 18/Output
//     PlcTask Outputs/GVL_iXlinker.EtherCAT_Master_EPPxxxx.Beckhoff_EPP2xxx.Beckhoff_EPP2xxxEK1122.A_0066_EPP2349_0021_0018.Channel_19.Output <-> Channel 19/Output
//     PlcTask Outputs/GVL_iXlinker.EtherCAT_Master_EPPxxxx.Beckhoff_EPP2xxx.Beckhoff_EPP2xxxEK1122.A_0066_EPP2349_0021_0018.Channel_20.Output <-> Channel 20/Output
//     PlcTask Outputs/GVL_iXlinker.EtherCAT_Master_EPPxxxx.Beckhoff_EPP2xxx.Beckhoff_EPP2xxxEK1122.A_0066_EPP2349_0021_0018.Channel_21.Output <-> Channel 21/Output
//     PlcTask Outputs/GVL_iXlinker.EtherCAT_Master_EPPxxxx.Beckhoff_EPP2xxx.Beckhoff_EPP2xxxEK1122.A_0066_EPP2349_0021_0018.Channel_22.Output <-> Channel 22/Output
//     PlcTask Outputs/GVL_iXlinker.EtherCAT_Master_EPPxxxx.Beckhoff_EPP2xxx.Beckhoff_EPP2xxxEK1122.A_0066_EPP2349_0021_0018.Channel_23.Output <-> Channel 23/Output
//     PlcTask Outputs/GVL_iXlinker.EtherCAT_Master_EPPxxxx.Beckhoff_EPP2xxx.Beckhoff_EPP2xxxEK1122.A_0066_EPP2349_0021_0018.Channel_24.Output <-> Channel 24/Output
//     PlcTask Outputs/GVL_iXlinker.EtherCAT_Master_EPPxxxx.Beckhoff_EPP2xxx.Beckhoff_EPP2xxxEK1122.A_0066_EPP2349_0021_0018.Channel_25.Output <-> Channel 25/Output
//     PlcTask Outputs/GVL_iXlinker.EtherCAT_Master_EPPxxxx.Beckhoff_EPP2xxx.Beckhoff_EPP2xxxEK1122.A_0066_EPP2349_0021_0018.Channel_26.Output <-> Channel 26/Output
//     PlcTask Outputs/GVL_iXlinker.EtherCAT_Master_EPPxxxx.Beckhoff_EPP2xxx.Beckhoff_EPP2xxxEK1122.A_0066_EPP2349_0021_0018.Channel_27.Output <-> Channel 27/Output
//     PlcTask Outputs/GVL_iXlinker.EtherCAT_Master_EPPxxxx.Beckhoff_EPP2xxx.Beckhoff_EPP2xxxEK1122.A_0066_EPP2349_0021_0018.Channel_28.Output <-> Channel 28/Output
//     PlcTask Outputs/GVL_iXlinker.EtherCAT_Master_EPPxxxx.Beckhoff_EPP2xxx.Beckhoff_EPP2xxxEK1122.A_0066_EPP2349_0021_0018.Channel_29.Output <-> Channel 29/Output
//     PlcTask Outputs/GVL_iXlinker.EtherCAT_Master_EPPxxxx.Beckhoff_EPP2xxx.Beckhoff_EPP2xxxEK1122.A_0066_EPP2349_0021_0018.Channel_30.Output <-> Channel 30/Output
//     PlcTask Outputs/GVL_iXlinker.EtherCAT_Master_EPPxxxx.Beckhoff_EPP2xxx.Beckhoff_EPP2xxxEK1122.A_0066_EPP2349_0021_0018.Channel_31.Output <-> Channel 31/Output
//     PlcTask Outputs/GVL_iXlinker.EtherCAT_Master_EPPxxxx.Beckhoff_EPP2xxx.Beckhoff_EPP2xxxEK1122.A_0066_EPP2349_0021_0018.Channel_32.Output <-> Channel 32/Output
//     PlcTask Inputs/GVL_iXlinker.EtherCAT_Master_EPPxxxx.Beckhoff_EPP2xxx.Beckhoff_EPP2xxxEK1122.A_0066_EPP2349_0021_0018.WcState.WcState <-> WcState/WcState
//     PlcTask Inputs/GVL_iXlinker.EtherCAT_Master_EPPxxxx.Beckhoff_EPP2xxx.Beckhoff_EPP2xxxEK1122.A_0066_EPP2349_0021_0018.WcState.InputToggle <-> WcState/InputToggle
//     PlcTask Inputs/GVL_iXlinker.EtherCAT_Master_EPPxxxx.Beckhoff_EPP2xxx.Beckhoff_EPP2xxxEK1122.A_0066_EPP2349_0021_0018.InfoData.State <-> InfoData/State
//   PLC/PLC Instance <-> EtherCAT Master EPPxxxx/Beckhoff EPP2xxx/Beckhoff EPP2xxxEK1122/A_0067(EPP2349-0022-0016)
//     PlcTask Inputs/GVL_iXlinker.EtherCAT_Master_EPPxxxx.Beckhoff_EPP2xxx.Beckhoff_EPP2xxxEK1122.A_0067_EPP2349_0022_0016.Channel_1.Input <-> Channel 1/Input
//     PlcTask Inputs/GVL_iXlinker.EtherCAT_Master_EPPxxxx.Beckhoff_EPP2xxx.Beckhoff_EPP2xxxEK1122.A_0067_EPP2349_0022_0016.Channel_2.Input <-> Channel 2/Input
//     PlcTask Inputs/GVL_iXlinker.EtherCAT_Master_EPPxxxx.Beckhoff_EPP2xxx.Beckhoff_EPP2xxxEK1122.A_0067_EPP2349_0022_0016.Channel_3.Input <-> Channel 3/Input
//     PlcTask Inputs/GVL_iXlinker.EtherCAT_Master_EPPxxxx.Beckhoff_EPP2xxx.Beckhoff_EPP2xxxEK1122.A_0067_EPP2349_0022_0016.Channel_4.Input <-> Channel 4/Input
//     PlcTask Inputs/GVL_iXlinker.EtherCAT_Master_EPPxxxx.Beckhoff_EPP2xxx.Beckhoff_EPP2xxxEK1122.A_0067_EPP2349_0022_0016.Channel_5.Input <-> Channel 5/Input
//     PlcTask Inputs/GVL_iXlinker.EtherCAT_Master_EPPxxxx.Beckhoff_EPP2xxx.Beckhoff_EPP2xxxEK1122.A_0067_EPP2349_0022_0016.Channel_6.Input <-> Channel 6/Input
//     PlcTask Inputs/GVL_iXlinker.EtherCAT_Master_EPPxxxx.Beckhoff_EPP2xxx.Beckhoff_EPP2xxxEK1122.A_0067_EPP2349_0022_0016.Channel_7.Input <-> Channel 7/Input
//     PlcTask Inputs/GVL_iXlinker.EtherCAT_Master_EPPxxxx.Beckhoff_EPP2xxx.Beckhoff_EPP2xxxEK1122.A_0067_EPP2349_0022_0016.Channel_8.Input <-> Channel 8/Input
//     PlcTask Inputs/GVL_iXlinker.EtherCAT_Master_EPPxxxx.Beckhoff_EPP2xxx.Beckhoff_EPP2xxxEK1122.A_0067_EPP2349_0022_0016.Channel_9.Input <-> Channel 9/Input
//     PlcTask Inputs/GVL_iXlinker.EtherCAT_Master_EPPxxxx.Beckhoff_EPP2xxx.Beckhoff_EPP2xxxEK1122.A_0067_EPP2349_0022_0016.Channel_10.Input <-> Channel 10/Input
//     PlcTask Inputs/GVL_iXlinker.EtherCAT_Master_EPPxxxx.Beckhoff_EPP2xxx.Beckhoff_EPP2xxxEK1122.A_0067_EPP2349_0022_0016.Channel_11.Input <-> Channel 11/Input
//     PlcTask Inputs/GVL_iXlinker.EtherCAT_Master_EPPxxxx.Beckhoff_EPP2xxx.Beckhoff_EPP2xxxEK1122.A_0067_EPP2349_0022_0016.Channel_12.Input <-> Channel 12/Input
//     PlcTask Inputs/GVL_iXlinker.EtherCAT_Master_EPPxxxx.Beckhoff_EPP2xxx.Beckhoff_EPP2xxxEK1122.A_0067_EPP2349_0022_0016.Channel_13.Input <-> Channel 13/Input
//     PlcTask Inputs/GVL_iXlinker.EtherCAT_Master_EPPxxxx.Beckhoff_EPP2xxx.Beckhoff_EPP2xxxEK1122.A_0067_EPP2349_0022_0016.Channel_14.Input <-> Channel 14/Input
//     PlcTask Inputs/GVL_iXlinker.EtherCAT_Master_EPPxxxx.Beckhoff_EPP2xxx.Beckhoff_EPP2xxxEK1122.A_0067_EPP2349_0022_0016.Channel_15.Input <-> Channel 15/Input
//     PlcTask Inputs/GVL_iXlinker.EtherCAT_Master_EPPxxxx.Beckhoff_EPP2xxx.Beckhoff_EPP2xxxEK1122.A_0067_EPP2349_0022_0016.Channel_16.Input <-> Channel 16/Input
//     PlcTask Outputs/GVL_iXlinker.EtherCAT_Master_EPPxxxx.Beckhoff_EPP2xxx.Beckhoff_EPP2xxxEK1122.A_0067_EPP2349_0022_0016.Channel_9_1.Output <-> Channel 9_1/Output
//     PlcTask Outputs/GVL_iXlinker.EtherCAT_Master_EPPxxxx.Beckhoff_EPP2xxx.Beckhoff_EPP2xxxEK1122.A_0067_EPP2349_0022_0016.Channel_10_1.Output <-> Channel 10_1/Output
//     PlcTask Outputs/GVL_iXlinker.EtherCAT_Master_EPPxxxx.Beckhoff_EPP2xxx.Beckhoff_EPP2xxxEK1122.A_0067_EPP2349_0022_0016.Channel_11_1.Output <-> Channel 11_1/Output
//     PlcTask Outputs/GVL_iXlinker.EtherCAT_Master_EPPxxxx.Beckhoff_EPP2xxx.Beckhoff_EPP2xxxEK1122.A_0067_EPP2349_0022_0016.Channel_12_1.Output <-> Channel 12_1/Output
//     PlcTask Outputs/GVL_iXlinker.EtherCAT_Master_EPPxxxx.Beckhoff_EPP2xxx.Beckhoff_EPP2xxxEK1122.A_0067_EPP2349_0022_0016.Channel_13_1.Output <-> Channel 13_1/Output
//     PlcTask Outputs/GVL_iXlinker.EtherCAT_Master_EPPxxxx.Beckhoff_EPP2xxx.Beckhoff_EPP2xxxEK1122.A_0067_EPP2349_0022_0016.Channel_14_1.Output <-> Channel 14_1/Output
//     PlcTask Outputs/GVL_iXlinker.EtherCAT_Master_EPPxxxx.Beckhoff_EPP2xxx.Beckhoff_EPP2xxxEK1122.A_0067_EPP2349_0022_0016.Channel_15_1.Output <-> Channel 15_1/Output
//     PlcTask Outputs/GVL_iXlinker.EtherCAT_Master_EPPxxxx.Beckhoff_EPP2xxx.Beckhoff_EPP2xxxEK1122.A_0067_EPP2349_0022_0016.Channel_16_1.Output <-> Channel 16_1/Output
//     PlcTask Outputs/GVL_iXlinker.EtherCAT_Master_EPPxxxx.Beckhoff_EPP2xxx.Beckhoff_EPP2xxxEK1122.A_0067_EPP2349_0022_0016.Channel_25.Output <-> Channel 25/Output
//     PlcTask Outputs/GVL_iXlinker.EtherCAT_Master_EPPxxxx.Beckhoff_EPP2xxx.Beckhoff_EPP2xxxEK1122.A_0067_EPP2349_0022_0016.Channel_26.Output <-> Channel 26/Output
//     PlcTask Outputs/GVL_iXlinker.EtherCAT_Master_EPPxxxx.Beckhoff_EPP2xxx.Beckhoff_EPP2xxxEK1122.A_0067_EPP2349_0022_0016.Channel_27.Output <-> Channel 27/Output
//     PlcTask Outputs/GVL_iXlinker.EtherCAT_Master_EPPxxxx.Beckhoff_EPP2xxx.Beckhoff_EPP2xxxEK1122.A_0067_EPP2349_0022_0016.Channel_28.Output <-> Channel 28/Output
//     PlcTask Outputs/GVL_iXlinker.EtherCAT_Master_EPPxxxx.Beckhoff_EPP2xxx.Beckhoff_EPP2xxxEK1122.A_0067_EPP2349_0022_0016.Channel_29.Output <-> Channel 29/Output
//     PlcTask Outputs/GVL_iXlinker.EtherCAT_Master_EPPxxxx.Beckhoff_EPP2xxx.Beckhoff_EPP2xxxEK1122.A_0067_EPP2349_0022_0016.Channel_30.Output <-> Channel 30/Output
//     PlcTask Outputs/GVL_iXlinker.EtherCAT_Master_EPPxxxx.Beckhoff_EPP2xxx.Beckhoff_EPP2xxxEK1122.A_0067_EPP2349_0022_0016.Channel_31.Output <-> Channel 31/Output
//     PlcTask Outputs/GVL_iXlinker.EtherCAT_Master_EPPxxxx.Beckhoff_EPP2xxx.Beckhoff_EPP2xxxEK1122.A_0067_EPP2349_0022_0016.Channel_32.Output <-> Channel 32/Output
//     PlcTask Inputs/GVL_iXlinker.EtherCAT_Master_EPPxxxx.Beckhoff_EPP2xxx.Beckhoff_EPP2xxxEK1122.A_0067_EPP2349_0022_0016.WcState.WcState <-> WcState/WcState
//     PlcTask Inputs/GVL_iXlinker.EtherCAT_Master_EPPxxxx.Beckhoff_EPP2xxx.Beckhoff_EPP2xxxEK1122.A_0067_EPP2349_0022_0016.WcState.InputToggle <-> WcState/InputToggle
//     PlcTask Inputs/GVL_iXlinker.EtherCAT_Master_EPPxxxx.Beckhoff_EPP2xxx.Beckhoff_EPP2xxxEK1122.A_0067_EPP2349_0022_0016.InfoData.State <-> InfoData/State
//   PLC/PLC Instance <-> EtherCAT Master EPPxxxx/Beckhoff EPP2xxx/Beckhoff EPP2xxxEK1122/A_0068(EPP2349-0022-0017)
//     PlcTask Inputs/GVL_iXlinker.EtherCAT_Master_EPPxxxx.Beckhoff_EPP2xxx.Beckhoff_EPP2xxxEK1122.A_0068_EPP2349_0022_0017.Channel_1.Input <-> Channel 1/Input
//     PlcTask Inputs/GVL_iXlinker.EtherCAT_Master_EPPxxxx.Beckhoff_EPP2xxx.Beckhoff_EPP2xxxEK1122.A_0068_EPP2349_0022_0017.Channel_2.Input <-> Channel 2/Input
//     PlcTask Inputs/GVL_iXlinker.EtherCAT_Master_EPPxxxx.Beckhoff_EPP2xxx.Beckhoff_EPP2xxxEK1122.A_0068_EPP2349_0022_0017.Channel_3.Input <-> Channel 3/Input
//     PlcTask Inputs/GVL_iXlinker.EtherCAT_Master_EPPxxxx.Beckhoff_EPP2xxx.Beckhoff_EPP2xxxEK1122.A_0068_EPP2349_0022_0017.Channel_4.Input <-> Channel 4/Input
//     PlcTask Inputs/GVL_iXlinker.EtherCAT_Master_EPPxxxx.Beckhoff_EPP2xxx.Beckhoff_EPP2xxxEK1122.A_0068_EPP2349_0022_0017.Channel_5.Input <-> Channel 5/Input
//     PlcTask Inputs/GVL_iXlinker.EtherCAT_Master_EPPxxxx.Beckhoff_EPP2xxx.Beckhoff_EPP2xxxEK1122.A_0068_EPP2349_0022_0017.Channel_6.Input <-> Channel 6/Input
//     PlcTask Inputs/GVL_iXlinker.EtherCAT_Master_EPPxxxx.Beckhoff_EPP2xxx.Beckhoff_EPP2xxxEK1122.A_0068_EPP2349_0022_0017.Channel_7.Input <-> Channel 7/Input
//     PlcTask Inputs/GVL_iXlinker.EtherCAT_Master_EPPxxxx.Beckhoff_EPP2xxx.Beckhoff_EPP2xxxEK1122.A_0068_EPP2349_0022_0017.Channel_8.Input <-> Channel 8/Input
//     PlcTask Inputs/GVL_iXlinker.EtherCAT_Master_EPPxxxx.Beckhoff_EPP2xxx.Beckhoff_EPP2xxxEK1122.A_0068_EPP2349_0022_0017.Channel_9.Input <-> Channel 9/Input
//     PlcTask Inputs/GVL_iXlinker.EtherCAT_Master_EPPxxxx.Beckhoff_EPP2xxx.Beckhoff_EPP2xxxEK1122.A_0068_EPP2349_0022_0017.Channel_10.Input <-> Channel 10/Input
//     PlcTask Inputs/GVL_iXlinker.EtherCAT_Master_EPPxxxx.Beckhoff_EPP2xxx.Beckhoff_EPP2xxxEK1122.A_0068_EPP2349_0022_0017.Channel_11.Input <-> Channel 11/Input
//     PlcTask Inputs/GVL_iXlinker.EtherCAT_Master_EPPxxxx.Beckhoff_EPP2xxx.Beckhoff_EPP2xxxEK1122.A_0068_EPP2349_0022_0017.Channel_12.Input <-> Channel 12/Input
//     PlcTask Inputs/GVL_iXlinker.EtherCAT_Master_EPPxxxx.Beckhoff_EPP2xxx.Beckhoff_EPP2xxxEK1122.A_0068_EPP2349_0022_0017.Channel_13.Input <-> Channel 13/Input
//     PlcTask Inputs/GVL_iXlinker.EtherCAT_Master_EPPxxxx.Beckhoff_EPP2xxx.Beckhoff_EPP2xxxEK1122.A_0068_EPP2349_0022_0017.Channel_14.Input <-> Channel 14/Input
//     PlcTask Inputs/GVL_iXlinker.EtherCAT_Master_EPPxxxx.Beckhoff_EPP2xxx.Beckhoff_EPP2xxxEK1122.A_0068_EPP2349_0022_0017.Channel_15.Input <-> Channel 15/Input
//     PlcTask Inputs/GVL_iXlinker.EtherCAT_Master_EPPxxxx.Beckhoff_EPP2xxx.Beckhoff_EPP2xxxEK1122.A_0068_EPP2349_0022_0017.Channel_16.Input <-> Channel 16/Input
//     PlcTask Outputs/GVL_iXlinker.EtherCAT_Master_EPPxxxx.Beckhoff_EPP2xxx.Beckhoff_EPP2xxxEK1122.A_0068_EPP2349_0022_0017.Channel_17.Output <-> Channel 17/Output
//     PlcTask Outputs/GVL_iXlinker.EtherCAT_Master_EPPxxxx.Beckhoff_EPP2xxx.Beckhoff_EPP2xxxEK1122.A_0068_EPP2349_0022_0017.Channel_18.Output <-> Channel 18/Output
//     PlcTask Outputs/GVL_iXlinker.EtherCAT_Master_EPPxxxx.Beckhoff_EPP2xxx.Beckhoff_EPP2xxxEK1122.A_0068_EPP2349_0022_0017.Channel_19.Output <-> Channel 19/Output
//     PlcTask Outputs/GVL_iXlinker.EtherCAT_Master_EPPxxxx.Beckhoff_EPP2xxx.Beckhoff_EPP2xxxEK1122.A_0068_EPP2349_0022_0017.Channel_20.Output <-> Channel 20/Output
//     PlcTask Outputs/GVL_iXlinker.EtherCAT_Master_EPPxxxx.Beckhoff_EPP2xxx.Beckhoff_EPP2xxxEK1122.A_0068_EPP2349_0022_0017.Channel_21.Output <-> Channel 21/Output
//     PlcTask Outputs/GVL_iXlinker.EtherCAT_Master_EPPxxxx.Beckhoff_EPP2xxx.Beckhoff_EPP2xxxEK1122.A_0068_EPP2349_0022_0017.Channel_22.Output <-> Channel 22/Output
//     PlcTask Outputs/GVL_iXlinker.EtherCAT_Master_EPPxxxx.Beckhoff_EPP2xxx.Beckhoff_EPP2xxxEK1122.A_0068_EPP2349_0022_0017.Channel_23.Output <-> Channel 23/Output
//     PlcTask Outputs/GVL_iXlinker.EtherCAT_Master_EPPxxxx.Beckhoff_EPP2xxx.Beckhoff_EPP2xxxEK1122.A_0068_EPP2349_0022_0017.Channel_24.Output <-> Channel 24/Output
//     PlcTask Outputs/GVL_iXlinker.EtherCAT_Master_EPPxxxx.Beckhoff_EPP2xxx.Beckhoff_EPP2xxxEK1122.A_0068_EPP2349_0022_0017.Channel_25.Output <-> Channel 25/Output
//     PlcTask Outputs/GVL_iXlinker.EtherCAT_Master_EPPxxxx.Beckhoff_EPP2xxx.Beckhoff_EPP2xxxEK1122.A_0068_EPP2349_0022_0017.Channel_26.Output <-> Channel 26/Output
//     PlcTask Outputs/GVL_iXlinker.EtherCAT_Master_EPPxxxx.Beckhoff_EPP2xxx.Beckhoff_EPP2xxxEK1122.A_0068_EPP2349_0022_0017.Channel_27.Output <-> Channel 27/Output
//     PlcTask Outputs/GVL_iXlinker.EtherCAT_Master_EPPxxxx.Beckhoff_EPP2xxx.Beckhoff_EPP2xxxEK1122.A_0068_EPP2349_0022_0017.Channel_28.Output <-> Channel 28/Output
//     PlcTask Outputs/GVL_iXlinker.EtherCAT_Master_EPPxxxx.Beckhoff_EPP2xxx.Beckhoff_EPP2xxxEK1122.A_0068_EPP2349_0022_0017.Channel_29.Output <-> Channel 29/Output
//     PlcTask Outputs/GVL_iXlinker.EtherCAT_Master_EPPxxxx.Beckhoff_EPP2xxx.Beckhoff_EPP2xxxEK1122.A_0068_EPP2349_0022_0017.Channel_30.Output <-> Channel 30/Output
//     PlcTask Outputs/GVL_iXlinker.EtherCAT_Master_EPPxxxx.Beckhoff_EPP2xxx.Beckhoff_EPP2xxxEK1122.A_0068_EPP2349_0022_0017.Channel_31.Output <-> Channel 31/Output
//     PlcTask Outputs/GVL_iXlinker.EtherCAT_Master_EPPxxxx.Beckhoff_EPP2xxx.Beckhoff_EPP2xxxEK1122.A_0068_EPP2349_0022_0017.Channel_32.Output <-> Channel 32/Output
//     PlcTask Inputs/GVL_iXlinker.EtherCAT_Master_EPPxxxx.Beckhoff_EPP2xxx.Beckhoff_EPP2xxxEK1122.A_0068_EPP2349_0022_0017.WcState.WcState <-> WcState/WcState
//     PlcTask Inputs/GVL_iXlinker.EtherCAT_Master_EPPxxxx.Beckhoff_EPP2xxx.Beckhoff_EPP2xxxEK1122.A_0068_EPP2349_0022_0017.WcState.InputToggle <-> WcState/InputToggle
//     PlcTask Inputs/GVL_iXlinker.EtherCAT_Master_EPPxxxx.Beckhoff_EPP2xxx.Beckhoff_EPP2xxxEK1122.A_0068_EPP2349_0022_0017.InfoData.State <-> InfoData/State
//   PLC/PLC Instance <-> EtherCAT Master EPPxxxx/Beckhoff EPP2xxx/Beckhoff EPP2xxxEK1122/A_0069(EPP2349-0022-0018)
//     PlcTask Inputs/GVL_iXlinker.EtherCAT_Master_EPPxxxx.Beckhoff_EPP2xxx.Beckhoff_EPP2xxxEK1122.A_0069_EPP2349_0022_0018.Channel_1.Input <-> Channel 1/Input
//     PlcTask Inputs/GVL_iXlinker.EtherCAT_Master_EPPxxxx.Beckhoff_EPP2xxx.Beckhoff_EPP2xxxEK1122.A_0069_EPP2349_0022_0018.Channel_2.Input <-> Channel 2/Input
//     PlcTask Inputs/GVL_iXlinker.EtherCAT_Master_EPPxxxx.Beckhoff_EPP2xxx.Beckhoff_EPP2xxxEK1122.A_0069_EPP2349_0022_0018.Channel_3.Input <-> Channel 3/Input
//     PlcTask Inputs/GVL_iXlinker.EtherCAT_Master_EPPxxxx.Beckhoff_EPP2xxx.Beckhoff_EPP2xxxEK1122.A_0069_EPP2349_0022_0018.Channel_4.Input <-> Channel 4/Input
//     PlcTask Inputs/GVL_iXlinker.EtherCAT_Master_EPPxxxx.Beckhoff_EPP2xxx.Beckhoff_EPP2xxxEK1122.A_0069_EPP2349_0022_0018.Channel_5.Input <-> Channel 5/Input
//     PlcTask Inputs/GVL_iXlinker.EtherCAT_Master_EPPxxxx.Beckhoff_EPP2xxx.Beckhoff_EPP2xxxEK1122.A_0069_EPP2349_0022_0018.Channel_6.Input <-> Channel 6/Input
//     PlcTask Inputs/GVL_iXlinker.EtherCAT_Master_EPPxxxx.Beckhoff_EPP2xxx.Beckhoff_EPP2xxxEK1122.A_0069_EPP2349_0022_0018.Channel_7.Input <-> Channel 7/Input
//     PlcTask Inputs/GVL_iXlinker.EtherCAT_Master_EPPxxxx.Beckhoff_EPP2xxx.Beckhoff_EPP2xxxEK1122.A_0069_EPP2349_0022_0018.Channel_8.Input <-> Channel 8/Input
//     PlcTask Inputs/GVL_iXlinker.EtherCAT_Master_EPPxxxx.Beckhoff_EPP2xxx.Beckhoff_EPP2xxxEK1122.A_0069_EPP2349_0022_0018.Channel_9.Input <-> Channel 9/Input
//     PlcTask Inputs/GVL_iXlinker.EtherCAT_Master_EPPxxxx.Beckhoff_EPP2xxx.Beckhoff_EPP2xxxEK1122.A_0069_EPP2349_0022_0018.Channel_10.Input <-> Channel 10/Input
//     PlcTask Inputs/GVL_iXlinker.EtherCAT_Master_EPPxxxx.Beckhoff_EPP2xxx.Beckhoff_EPP2xxxEK1122.A_0069_EPP2349_0022_0018.Channel_11.Input <-> Channel 11/Input
//     PlcTask Inputs/GVL_iXlinker.EtherCAT_Master_EPPxxxx.Beckhoff_EPP2xxx.Beckhoff_EPP2xxxEK1122.A_0069_EPP2349_0022_0018.Channel_12.Input <-> Channel 12/Input
//     PlcTask Inputs/GVL_iXlinker.EtherCAT_Master_EPPxxxx.Beckhoff_EPP2xxx.Beckhoff_EPP2xxxEK1122.A_0069_EPP2349_0022_0018.Channel_13.Input <-> Channel 13/Input
//     PlcTask Inputs/GVL_iXlinker.EtherCAT_Master_EPPxxxx.Beckhoff_EPP2xxx.Beckhoff_EPP2xxxEK1122.A_0069_EPP2349_0022_0018.Channel_14.Input <-> Channel 14/Input
//     PlcTask Inputs/GVL_iXlinker.EtherCAT_Master_EPPxxxx.Beckhoff_EPP2xxx.Beckhoff_EPP2xxxEK1122.A_0069_EPP2349_0022_0018.Channel_15.Input <-> Channel 15/Input
//     PlcTask Inputs/GVL_iXlinker.EtherCAT_Master_EPPxxxx.Beckhoff_EPP2xxx.Beckhoff_EPP2xxxEK1122.A_0069_EPP2349_0022_0018.Channel_16.Input <-> Channel 16/Input
//     PlcTask Outputs/GVL_iXlinker.EtherCAT_Master_EPPxxxx.Beckhoff_EPP2xxx.Beckhoff_EPP2xxxEK1122.A_0069_EPP2349_0022_0018.Channel_17.Output <-> Channel 17/Output
//     PlcTask Outputs/GVL_iXlinker.EtherCAT_Master_EPPxxxx.Beckhoff_EPP2xxx.Beckhoff_EPP2xxxEK1122.A_0069_EPP2349_0022_0018.Channel_18.Output <-> Channel 18/Output
//     PlcTask Outputs/GVL_iXlinker.EtherCAT_Master_EPPxxxx.Beckhoff_EPP2xxx.Beckhoff_EPP2xxxEK1122.A_0069_EPP2349_0022_0018.Channel_19.Output <-> Channel 19/Output
//     PlcTask Outputs/GVL_iXlinker.EtherCAT_Master_EPPxxxx.Beckhoff_EPP2xxx.Beckhoff_EPP2xxxEK1122.A_0069_EPP2349_0022_0018.Channel_20.Output <-> Channel 20/Output
//     PlcTask Outputs/GVL_iXlinker.EtherCAT_Master_EPPxxxx.Beckhoff_EPP2xxx.Beckhoff_EPP2xxxEK1122.A_0069_EPP2349_0022_0018.Channel_21.Output <-> Channel 21/Output
//     PlcTask Outputs/GVL_iXlinker.EtherCAT_Master_EPPxxxx.Beckhoff_EPP2xxx.Beckhoff_EPP2xxxEK1122.A_0069_EPP2349_0022_0018.Channel_22.Output <-> Channel 22/Output
//     PlcTask Outputs/GVL_iXlinker.EtherCAT_Master_EPPxxxx.Beckhoff_EPP2xxx.Beckhoff_EPP2xxxEK1122.A_0069_EPP2349_0022_0018.Channel_23.Output <-> Channel 23/Output
//     PlcTask Outputs/GVL_iXlinker.EtherCAT_Master_EPPxxxx.Beckhoff_EPP2xxx.Beckhoff_EPP2xxxEK1122.A_0069_EPP2349_0022_0018.Channel_24.Output <-> Channel 24/Output
//     PlcTask Outputs/GVL_iXlinker.EtherCAT_Master_EPPxxxx.Beckhoff_EPP2xxx.Beckhoff_EPP2xxxEK1122.A_0069_EPP2349_0022_0018.Channel_25.Output <-> Channel 25/Output
//     PlcTask Outputs/GVL_iXlinker.EtherCAT_Master_EPPxxxx.Beckhoff_EPP2xxx.Beckhoff_EPP2xxxEK1122.A_0069_EPP2349_0022_0018.Channel_26.Output <-> Channel 26/Output
//     PlcTask Outputs/GVL_iXlinker.EtherCAT_Master_EPPxxxx.Beckhoff_EPP2xxx.Beckhoff_EPP2xxxEK1122.A_0069_EPP2349_0022_0018.Channel_27.Output <-> Channel 27/Output
//     PlcTask Outputs/GVL_iXlinker.EtherCAT_Master_EPPxxxx.Beckhoff_EPP2xxx.Beckhoff_EPP2xxxEK1122.A_0069_EPP2349_0022_0018.Channel_28.Output <-> Channel 28/Output
//     PlcTask Outputs/GVL_iXlinker.EtherCAT_Master_EPPxxxx.Beckhoff_EPP2xxx.Beckhoff_EPP2xxxEK1122.A_0069_EPP2349_0022_0018.Channel_29.Output <-> Channel 29/Output
//     PlcTask Outputs/GVL_iXlinker.EtherCAT_Master_EPPxxxx.Beckhoff_EPP2xxx.Beckhoff_EPP2xxxEK1122.A_0069_EPP2349_0022_0018.Channel_30.Output <-> Channel 30/Output
//     PlcTask Outputs/GVL_iXlinker.EtherCAT_Master_EPPxxxx.Beckhoff_EPP2xxx.Beckhoff_EPP2xxxEK1122.A_0069_EPP2349_0022_0018.Channel_31.Output <-> Channel 31/Output
//     PlcTask Outputs/GVL_iXlinker.EtherCAT_Master_EPPxxxx.Beckhoff_EPP2xxx.Beckhoff_EPP2xxxEK1122.A_0069_EPP2349_0022_0018.Channel_32.Output <-> Channel 32/Output
//     PlcTask Inputs/GVL_iXlinker.EtherCAT_Master_EPPxxxx.Beckhoff_EPP2xxx.Beckhoff_EPP2xxxEK1122.A_0069_EPP2349_0022_0018.WcState.WcState <-> WcState/WcState
//     PlcTask Inputs/GVL_iXlinker.EtherCAT_Master_EPPxxxx.Beckhoff_EPP2xxx.Beckhoff_EPP2xxxEK1122.A_0069_EPP2349_0022_0018.WcState.InputToggle <-> WcState/InputToggle
//     PlcTask Inputs/GVL_iXlinker.EtherCAT_Master_EPPxxxx.Beckhoff_EPP2xxx.Beckhoff_EPP2xxxEK1122.A_0069_EPP2349_0022_0018.InfoData.State <-> InfoData/State
//   PLC/PLC Instance <-> EtherCAT Master EPPxxxx/Beckhoff EPP2xxx/Beckhoff EPP2xxxEK1122/A_0070(EPP2624-0002-0016)
//     PlcTask Outputs/GVL_iXlinker.EtherCAT_Master_EPPxxxx.Beckhoff_EPP2xxx.Beckhoff_EPP2xxxEK1122.A_0070_EPP2624_0002_0016.Channel_1.Output <-> Channel 1/Output
//     PlcTask Outputs/GVL_iXlinker.EtherCAT_Master_EPPxxxx.Beckhoff_EPP2xxx.Beckhoff_EPP2xxxEK1122.A_0070_EPP2624_0002_0016.Channel_2.Output <-> Channel 2/Output
//     PlcTask Outputs/GVL_iXlinker.EtherCAT_Master_EPPxxxx.Beckhoff_EPP2xxx.Beckhoff_EPP2xxxEK1122.A_0070_EPP2624_0002_0016.Channel_3.Output <-> Channel 3/Output
//     PlcTask Outputs/GVL_iXlinker.EtherCAT_Master_EPPxxxx.Beckhoff_EPP2xxx.Beckhoff_EPP2xxxEK1122.A_0070_EPP2624_0002_0016.Channel_4.Output <-> Channel 4/Output
//     PlcTask Inputs/GVL_iXlinker.EtherCAT_Master_EPPxxxx.Beckhoff_EPP2xxx.Beckhoff_EPP2xxxEK1122.A_0070_EPP2624_0002_0016.WcState.WcState <-> WcState/WcState
//     PlcTask Inputs/GVL_iXlinker.EtherCAT_Master_EPPxxxx.Beckhoff_EPP2xxx.Beckhoff_EPP2xxxEK1122.A_0070_EPP2624_0002_0016.InfoData.State <-> InfoData/State
//   PLC/PLC Instance <-> EtherCAT Master EPPxxxx/Beckhoff EPP2xxx/Beckhoff EPP2xxxEK1122/A_0071(EPP2809-0021-0016)
//     PlcTask Outputs/GVL_iXlinker.EtherCAT_Master_EPPxxxx.Beckhoff_EPP2xxx.Beckhoff_EPP2xxxEK1122.A_0071_EPP2809_0021_0016.Channel_1.Output <-> Channel 1/Output
//     PlcTask Outputs/GVL_iXlinker.EtherCAT_Master_EPPxxxx.Beckhoff_EPP2xxx.Beckhoff_EPP2xxxEK1122.A_0071_EPP2809_0021_0016.Channel_2.Output <-> Channel 2/Output
//     PlcTask Outputs/GVL_iXlinker.EtherCAT_Master_EPPxxxx.Beckhoff_EPP2xxx.Beckhoff_EPP2xxxEK1122.A_0071_EPP2809_0021_0016.Channel_3.Output <-> Channel 3/Output
//     PlcTask Outputs/GVL_iXlinker.EtherCAT_Master_EPPxxxx.Beckhoff_EPP2xxx.Beckhoff_EPP2xxxEK1122.A_0071_EPP2809_0021_0016.Channel_4.Output <-> Channel 4/Output
